  PROC DrawPart84()
    MoveL Offs(pOrigin,162.64,96.16,0.00),v40,z0,tPen\WObj:=wPaper;
    MoveL Offs(pOrigin,162.24,96.31,0.00),v40,z0,tPen\WObj:=wPaper;
    MoveL Offs(pOrigin,173.08,96.31,0.00),v40,z0,tPen\WObj:=wPaper;
    MoveL Offs(pOrigin,173.29,96.59,0.00),v40,z0,tPen\WObj:=wPaper;
    MoveL Offs(pOrigin,180.51,104.24,0.00),v40,z0,tPen\WObj:=wPaper;
    MoveL Offs(pOrigin,193.05,116.56,0.00),v40,fine,tPen\WObj:=wPaper;
    MoveL Offs(pOrigin,193.05,116.56,6.00),v60,z5,tPen\WObj:=wPaper;
    MoveL Offs(pOrigin,193.92,115.46,6.00),vTravel,z5,tPen\WObj:=wPaper;
    MoveL Offs(pOrigin,193.92,115.46,0.00),v60,z0,tPen\WObj:=wPaper;
    MoveL Offs(pOrigin,194.97,114.41,0.00),v40,z0,tPen\WObj:=wPaper;
    MoveL Offs(pOrigin,195.87,115.01,0.00),v40,z0,tPen\WObj:=wPaper;
    MoveL Offs(pOrigin,194.82,116.06,0.00),v40,z0,tPen\WObj:=wPaper;
    MoveL Offs(pOrigin,195.71,116.66,0.00),v40,z0,tPen\WObj:=wPaper;
    MoveL Offs(pOrigin,196.47,115.91,0.00),v40,fine,tPen\WObj:=wPaper;
    MoveL Offs(pOrigin,196.47,115.91,6.00),v60,z5,tPen\WObj:=wPaper;
    MoveL Offs(pOrigin,194.38,113.52,6.00),vTravel,z5,tPen\WObj:=wPaper;
    MoveL Offs(pOrigin,194.38,113.52,0.00),v60,z0,tPen\WObj:=wPaper;
    MoveL Offs(pOrigin,193.02,114.87,0.00),v40,z0,tPen\WObj:=wPaper;
    MoveL Offs(pOrigin,193.69,114.22,0.00),v40,z0,tPen\WObj:=wPaper;
    MoveL Offs(pOrigin,194.11,114.65,0.00),v40,z0,tPen\WObj:=wPaper;
    MoveL Offs(pOrigin,193.69,114.22,0.00),v40,fine,tPen\WObj:=wPaper;
    MoveL Offs(pOrigin,193.69,114.22,6.00),v60,z5,tPen\WObj:=wPaper;
    MoveL Offs(pOrigin,193.48,112.92,6.00),vTravel,z5,tPen\WObj:=wPaper;
    MoveL Offs(pOrigin,193.48,112.92,0.00),v60,z0,tPen\WObj:=wPaper;
    MoveL Offs(pOrigin,191.68,114.72,0.00),v40,z0,tPen\WObj:=wPaper;
    MoveL Offs(pOrigin,190.63,114.28,0.00),v40,z0,tPen\WObj:=wPaper;
    MoveL Offs(pOrigin,192.88,112.02,0.00),v40,z0,tPen\WObj:=wPaper;
    MoveL Offs(pOrigin,191.99,111.43,0.00),v40,z0,tPen\WObj:=wPaper;
    MoveL Offs(pOrigin,189.88,113.53,0.00),v40,z0,tPen\WObj:=wPaper;
    MoveL Offs(pOrigin,188.98,112.93,0.00),v40,z0,tPen\WObj:=wPaper;
    MoveL Offs(pOrigin,191.39,110.53,0.00),v40,z0,tPen\WObj:=wPaper;
    MoveL Offs(pOrigin,190.64,109.78,0.00),v40,z0,tPen\WObj:=wPaper;
    MoveL Offs(pOrigin,188.09,112.34,0.00),v40,z0,tPen\WObj:=wPaper;
    MoveL Offs(pOrigin,187.34,111.59,0.00),v40,z0,tPen\WObj:=wPaper;
    MoveL Offs(pOrigin,189.90,109.04,0.00),v40,z0,tPen\WObj:=wPaper;
    MoveL Offs(pOrigin,189.15,108.29,0.00),v40,z0,tPen\WObj:=wPaper;
    MoveL Offs(pOrigin,186.44,110.99,0.00),v40,z0,tPen\WObj:=wPaper;
    MoveL Offs(pOrigin,186.46,109.97,0.00),v40,z0,tPen\WObj:=wPaper;
    MoveL Offs(pOrigin,186.89,110.40,0.00),v40,z0,tPen\WObj:=wPaper;
    MoveL Offs(pOrigin,186.46,109.97,0.00),v40,z0,tPen\WObj:=wPaper;
    MoveL Offs(pOrigin,185.70,110.25,0.00),v40,z0,tPen\WObj:=wPaper;
    MoveL Offs(pOrigin,188.55,107.39,0.00),v40,z0,tPen\WObj:=wPaper;
    MoveL Offs(pOrigin,187.81,106.65,0.00),v40,z0,tPen\WObj:=wPaper;
    MoveL Offs(pOrigin,184.95,109.50,0.00),v40,z0,tPen\WObj:=wPaper;
    MoveL Offs(pOrigin,184.20,108.75,0.00),v40,z0,tPen\WObj:=wPaper;
    MoveL Offs(pOrigin,187.21,105.75,0.00),v40,z0,tPen\WObj:=wPaper;
    MoveL Offs(pOrigin,186.46,105.00,0.00),v40,z0,tPen\WObj:=wPaper;
    MoveL Offs(pOrigin,183.31,108.16,0.00),v40,z0,tPen\WObj:=wPaper;
    MoveL Offs(pOrigin,183.70,107.21,0.00),v40,z0,tPen\WObj:=wPaper;
    MoveL Offs(pOrigin,184.55,108.06,0.00),v40,z0,tPen\WObj:=wPaper;
    MoveL Offs(pOrigin,183.70,107.21,0.00),v40,z0,tPen\WObj:=wPaper;
    MoveL Offs(pOrigin,182.71,107.26,0.00),v40,z0,tPen\WObj:=wPaper;
    MoveL Offs(pOrigin,185.87,104.10,0.00),v40,z0,tPen\WObj:=wPaper;
    MoveL Offs(pOrigin,185.27,103.21,0.00),v40,z0,tPen\WObj:=wPaper;
    MoveL Offs(pOrigin,181.81,106.66,0.00),v40,z0,tPen\WObj:=wPaper;
    MoveL Offs(pOrigin,182.21,105.72,0.00),v40,z0,tPen\WObj:=wPaper;
    MoveL Offs(pOrigin,183.06,106.57,0.00),v40,z0,tPen\WObj:=wPaper;
    MoveL Offs(pOrigin,182.21,105.72,0.00),v40,z0,tPen\WObj:=wPaper;
    MoveL Offs(pOrigin,181.07,105.92,0.00),v40,z0,tPen\WObj:=wPaper;
    MoveL Offs(pOrigin,182.42,104.56,0.00),v40,z0,tPen\WObj:=wPaper;
    MoveL Offs(pOrigin,181.67,103.82,0.00),v40,z0,tPen\WObj:=wPaper;
    MoveL Offs(pOrigin,180.32,105.17,0.00),v40,z0,tPen\WObj:=wPaper;
    MoveL Offs(pOrigin,181.15,104.66,0.00),v40,z0,tPen\WObj:=wPaper;
    MoveL Offs(pOrigin,182.00,105.51,0.00),v40,z0,tPen\WObj:=wPaper;
    MoveL Offs(pOrigin,181.15,104.66,0.00),v40,fine,tPen\WObj:=wPaper;
    MoveL Offs(pOrigin,181.15,104.66,6.00),v60,z5,tPen\WObj:=wPaper;
    MoveL Offs(pOrigin,179.57,104.42,6.00),vTravel,z5,tPen\WObj:=wPaper;
    MoveL Offs(pOrigin,179.57,104.42,0.00),v60,z0,tPen\WObj:=wPaper;
    MoveL Offs(pOrigin,180.93,103.07,0.00),v40,z0,tPen\WObj:=wPaper;
    MoveL Offs(pOrigin,180.18,102.32,0.00),v40,z0,tPen\WObj:=wPaper;
    MoveL Offs(pOrigin,178.83,103.68,0.00),v40,z0,tPen\WObj:=wPaper;
    MoveL Offs(pOrigin,179.59,103.72,0.00),v40,z0,tPen\WObj:=wPaper;
    MoveL Offs(pOrigin,175.68,99.81,0.00),v40,z0,tPen\WObj:=wPaper;
    MoveL Offs(pOrigin,175.09,99.94,0.00),v40,z0,tPen\WObj:=wPaper;
    MoveL Offs(pOrigin,176.60,98.44,0.00),v40,z0,tPen\WObj:=wPaper;
    MoveL Offs(pOrigin,175.84,99.14,0.00),v40,z0,tPen\WObj:=wPaper;
    MoveL Offs(pOrigin,176.26,99.56,0.00),v40,z0,tPen\WObj:=wPaper;
    MoveL Offs(pOrigin,175.84,99.14,0.00),v40,fine,tPen\WObj:=wPaper;
    MoveL Offs(pOrigin,175.84,99.14,6.00),v60,z5,tPen\WObj:=wPaper;
    MoveL Offs(pOrigin,174.50,99.05,6.00),vTravel,z5,tPen\WObj:=wPaper;
    MoveL Offs(pOrigin,174.50,99.05,0.00),v60,z0,tPen\WObj:=wPaper;
    MoveL Offs(pOrigin,175.85,97.69,0.00),v40,z0,tPen\WObj:=wPaper;
    MoveL Offs(pOrigin,175.10,96.95,0.00),v40,z0,tPen\WObj:=wPaper;
    MoveL Offs(pOrigin,173.60,98.45,0.00),v40,z0,tPen\WObj:=wPaper;
    MoveL Offs(pOrigin,173.00,97.55,0.00),v40,z0,tPen\WObj:=wPaper;
    MoveL Offs(pOrigin,202.60,67.95,0.00),v40,z0,tPen\WObj:=wPaper;
    MoveL Offs(pOrigin,203.75,68.14,0.00),v40,z0,tPen\WObj:=wPaper;
    MoveL Offs(pOrigin,205.55,69.94,0.00),v40,z0,tPen\WObj:=wPaper;
    MoveL Offs(pOrigin,205.80,69.60,0.00),v40,z0,tPen\WObj:=wPaper;
    MoveL Offs(pOrigin,206.23,68.75,0.00),v40,z0,tPen\WObj:=wPaper;
    MoveL Offs(pOrigin,214.51,62.52,0.00),v40,z0,tPen\WObj:=wPaper;
    MoveL Offs(pOrigin,214.73,63.22,0.00),v40,z0,tPen\WObj:=wPaper;
    MoveL Offs(pOrigin,214.30,68.96,0.00),v40,z0,tPen\WObj:=wPaper;
    MoveL Offs(pOrigin,213.95,70.24,0.00),v40,z0,tPen\WObj:=wPaper;
    MoveL Offs(pOrigin,213.02,71.51,0.00),v40,z0,tPen\WObj:=wPaper;
    MoveL Offs(pOrigin,212.59,71.01,0.00),v40,z0,tPen\WObj:=wPaper;
    MoveL Offs(pOrigin,214.40,72.82,0.00),v40,z0,tPen\WObj:=wPaper;
    MoveL Offs(pOrigin,214.09,72.57,0.00),v40,z0,tPen\WObj:=wPaper;
    MoveL Offs(pOrigin,215.01,71.30,0.00),v40,z0,tPen\WObj:=wPaper;
    MoveL Offs(pOrigin,215.86,68.61,0.00),v40,z0,tPen\WObj:=wPaper;
    MoveL Offs(pOrigin,216.21,68.54,0.00),v40,z0,tPen\WObj:=wPaper;
    MoveL Offs(pOrigin,216.21,68.54,0.00),v40,z0,tPen\WObj:=wPaper;
    MoveL Offs(pOrigin,216.00,64.93,0.00),v40,z0,tPen\WObj:=wPaper;
    MoveL Offs(pOrigin,216.21,63.86,0.00),v40,fine,tPen\WObj:=wPaper;
    MoveL Offs(pOrigin,216.21,63.86,6.00),v60,z5,tPen\WObj:=wPaper;
    MoveL Offs(pOrigin,217.49,63.58,6.00),vTravel,z5,tPen\WObj:=wPaper;
    MoveL Offs(pOrigin,217.49,63.58,0.00),v60,z0,tPen\WObj:=wPaper;
    MoveL Offs(pOrigin,214.51,63.58,0.00),v40,z0,tPen\WObj:=wPaper;
    MoveL Offs(pOrigin,214.38,62.59,0.00),v40,z0,tPen\WObj:=wPaper;
    MoveL Offs(pOrigin,214.38,60.89,0.00),v40,z0,tPen\WObj:=wPaper;
    MoveL Offs(pOrigin,214.30,60.46,0.00),v40,z0,tPen\WObj:=wPaper;
    MoveL Offs(pOrigin,213.24,61.53,0.00),v40,z0,tPen\WObj:=wPaper;
    MoveL Offs(pOrigin,214.30,60.46,0.00),v40,z0,tPen\WObj:=wPaper;
    MoveL Offs(pOrigin,214.51,60.41,0.00),v40,z0,tPen\WObj:=wPaper;
    MoveL Offs(pOrigin,217.28,60.41,0.00),v40,z0,tPen\WObj:=wPaper;
    MoveL Offs(pOrigin,218.06,59.96,0.00),v40,z0,tPen\WObj:=wPaper;
    MoveL Offs(pOrigin,212.95,65.07,0.00),v40,z0,tPen\WObj:=wPaper;
    MoveL Offs(pOrigin,212.12,64.57,0.00),v40,z0,tPen\WObj:=wPaper;
    MoveL Offs(pOrigin,210.77,63.22,0.00),v40,z0,tPen\WObj:=wPaper;
    MoveL Offs(pOrigin,211.11,63.58,0.00),v40,z0,tPen\WObj:=wPaper;
  ENDPROC

  PROC DrawPart85()
    MoveL Offs(pOrigin,212.60,63.58,0.00),v40,z0,tPen\WObj:=wPaper;
    MoveL Offs(pOrigin,212.39,62.52,0.00),v40,z0,tPen\WObj:=wPaper;
    MoveL Offs(pOrigin,217.49,62.52,0.00),v40,z0,tPen\WObj:=wPaper;
    MoveL Offs(pOrigin,217.96,62.94,0.00),v40,z0,tPen\WObj:=wPaper;
    MoveL Offs(pOrigin,214.51,59.48,0.00),v40,z0,tPen\WObj:=wPaper;
    MoveL Offs(pOrigin,214.94,59.19,0.00),v40,z0,tPen\WObj:=wPaper;
    MoveL Offs(pOrigin,213.66,58.76,0.00),v40,z0,tPen\WObj:=wPaper;
    MoveL Offs(pOrigin,212.46,56.64,0.00),v40,z0,tPen\WObj:=wPaper;
    MoveL Offs(pOrigin,212.18,54.72,0.00),v40,z0,tPen\WObj:=wPaper;
    MoveL Offs(pOrigin,212.60,53.88,0.00),v40,z0,tPen\WObj:=wPaper;
    MoveL Offs(pOrigin,212.99,53.49,0.00),v40,z0,tPen\WObj:=wPaper;
    MoveL Offs(pOrigin,211.04,51.53,0.00),v40,z0,tPen\WObj:=wPaper;
    MoveL Offs(pOrigin,211.32,51.96,0.00),v40,z0,tPen\WObj:=wPaper;
    MoveL Offs(pOrigin,215.58,51.96,0.00),v40,fine,tPen\WObj:=wPaper;
    MoveL Offs(pOrigin,215.58,51.96,6.00),v60,z5,tPen\WObj:=wPaper;
    MoveL Offs(pOrigin,216.49,52.81,6.00),vTravel,z5,tPen\WObj:=wPaper;
    MoveL Offs(pOrigin,216.49,52.81,0.00),v60,z0,tPen\WObj:=wPaper;
    MoveL Offs(pOrigin,216.49,54.30,0.00),v40,z0,tPen\WObj:=wPaper;
    MoveL Offs(pOrigin,215.79,54.07,0.00),v40,z0,tPen\WObj:=wPaper;
    MoveL Offs(pOrigin,218.12,54.07,0.00),v40,z0,tPen\WObj:=wPaper;
    MoveL Offs(pOrigin,217.55,53.88,0.00),v40,z0,tPen\WObj:=wPaper;
    MoveL Offs(pOrigin,217.55,52.60,0.00),v40,z0,tPen\WObj:=wPaper;
    MoveL Offs(pOrigin,217.28,51.96,0.00),v40,z0,tPen\WObj:=wPaper;
    MoveL Offs(pOrigin,219.82,51.96,0.00),v40,z0,tPen\WObj:=wPaper;
    MoveL Offs(pOrigin,219.61,52.17,0.00),v40,z0,tPen\WObj:=wPaper;
    MoveL Offs(pOrigin,219.19,52.60,0.00),v40,z0,tPen\WObj:=wPaper;
    MoveL Offs(pOrigin,219.61,52.17,0.00),v40,z0,tPen\WObj:=wPaper;
    MoveL Offs(pOrigin,219.73,52.76,0.00),v40,z0,tPen\WObj:=wPaper;
    MoveL Offs(pOrigin,217.77,50.81,0.00),v40,z0,tPen\WObj:=wPaper;
    MoveL Offs(pOrigin,218.34,50.90,0.00),v40,z0,tPen\WObj:=wPaper;
    MoveL Offs(pOrigin,222.80,50.90,0.00),v40,z0,tPen\WObj:=wPaper;
    MoveL Offs(pOrigin,223.01,50.07,0.00),v40,z0,tPen\WObj:=wPaper;
    MoveL Offs(pOrigin,220.61,47.67,0.00),v40,z0,tPen\WObj:=wPaper;
    MoveL Offs(pOrigin,221.31,47.74,0.00),v40,z0,tPen\WObj:=wPaper;
    MoveL Offs(pOrigin,223.22,47.74,0.00),v40,z0,tPen\WObj:=wPaper;
    MoveL Offs(pOrigin,223.44,47.71,0.00),v40,z0,tPen\WObj:=wPaper;
    MoveL Offs(pOrigin,223.01,48.35,0.00),v40,z0,tPen\WObj:=wPaper;
    MoveL Offs(pOrigin,223.44,47.71,0.00),v40,z0,tPen\WObj:=wPaper;
    MoveL Offs(pOrigin,223.76,47.83,0.00),v40,z0,tPen\WObj:=wPaper;
    MoveL Offs(pOrigin,216.54,40.62,0.00),v40,z0,tPen\WObj:=wPaper;
    MoveL Offs(pOrigin,215.57,40.05,0.00),v40,z0,tPen\WObj:=wPaper;
    MoveL Offs(pOrigin,211.52,44.11,0.00),v40,z0,tPen\WObj:=wPaper;
    MoveL Offs(pOrigin,210.56,43.59,0.00),v40,z0,tPen\WObj:=wPaper;
    MoveL Offs(pOrigin,199.59,32.62,0.00),v40,z0,tPen\WObj:=wPaper;
    MoveL Offs(pOrigin,200.06,32.95,0.00),v40,z0,tPen\WObj:=wPaper;
    MoveL Offs(pOrigin,195.39,32.95,0.00),v40,fine,tPen\WObj:=wPaper;
    MoveL Offs(pOrigin,195.39,32.95,6.00),v60,z5,tPen\WObj:=wPaper;
    MoveL Offs(pOrigin,196.02,31.90,6.00),vTravel,z5,tPen\WObj:=wPaper;
    MoveL Offs(pOrigin,196.02,31.90,0.00),v60,z0,tPen\WObj:=wPaper;
    MoveL Offs(pOrigin,166.70,31.90,0.00),v40,z0,tPen\WObj:=wPaper;
    MoveL Offs(pOrigin,167.23,31.63,0.00),v40,z0,tPen\WObj:=wPaper;
    MoveL Offs(pOrigin,168.89,33.28,0.00),v40,z0,tPen\WObj:=wPaper;
    MoveL Offs(pOrigin,168.11,33.75,0.00),v40,z0,tPen\WObj:=wPaper;
    MoveL Offs(pOrigin,171.11,30.75,0.00),v40,z0,tPen\WObj:=wPaper;
    MoveL Offs(pOrigin,171.28,31.19,0.00),v40,z0,tPen\WObj:=wPaper;
    MoveL Offs(pOrigin,173.08,32.99,0.00),v40,z0,tPen\WObj:=wPaper;
    MoveL Offs(pOrigin,172.90,33.44,0.00),v40,z0,tPen\WObj:=wPaper;
    MoveL Offs(pOrigin,175.61,30.73,0.00),v40,z0,tPen\WObj:=wPaper;
    MoveL Offs(pOrigin,175.62,31.05,0.00),v40,z0,tPen\WObj:=wPaper;
    MoveL Offs(pOrigin,177.87,33.31,0.00),v40,z0,tPen\WObj:=wPaper;
    MoveL Offs(pOrigin,176.94,33.88,0.00),v40,z0,tPen\WObj:=wPaper;
    MoveL Offs(pOrigin,180.10,30.72,0.00),v40,z0,tPen\WObj:=wPaper;
    MoveL Offs(pOrigin,180.41,31.37,0.00),v40,z0,tPen\WObj:=wPaper;
    MoveL Offs(pOrigin,181.92,32.87,0.00),v40,z0,tPen\WObj:=wPaper;
    MoveL Offs(pOrigin,182.04,33.26,0.00),v40,z0,tPen\WObj:=wPaper;
    MoveL Offs(pOrigin,184.89,30.41,0.00),v40,z0,tPen\WObj:=wPaper;
    MoveL Offs(pOrigin,184.46,30.93,0.00),v40,z0,tPen\WObj:=wPaper;
    MoveL Offs(pOrigin,186.26,32.73,0.00),v40,z0,tPen\WObj:=wPaper;
    MoveL Offs(pOrigin,186.53,33.25,0.00),v40,z0,tPen\WObj:=wPaper;
    MoveL Offs(pOrigin,189.39,30.39,0.00),v40,z0,tPen\WObj:=wPaper;
    MoveL Offs(pOrigin,188.95,30.94,0.00),v40,z0,tPen\WObj:=wPaper;
    MoveL Offs(pOrigin,190.90,32.90,0.00),v40,z0,tPen\WObj:=wPaper;
    MoveL Offs(pOrigin,191.03,33.23,0.00),v40,z0,tPen\WObj:=wPaper;
    MoveL Offs(pOrigin,193.58,30.68,0.00),v40,z0,tPen\WObj:=wPaper;
    MoveL Offs(pOrigin,193.90,31.41,0.00),v40,z0,tPen\WObj:=wPaper;
    MoveL Offs(pOrigin,199.91,37.42,0.00),v40,z0,tPen\WObj:=wPaper;
    MoveL Offs(pOrigin,199.85,37.85,0.00),v40,z0,tPen\WObj:=wPaper;
    MoveL Offs(pOrigin,205.86,31.84,0.00),v40,fine,tPen\WObj:=wPaper;
    MoveL Offs(pOrigin,205.86,31.84,6.00),v60,z5,tPen\WObj:=wPaper;
    MoveL Offs(pOrigin,204.36,31.84,6.00),vTravel,z5,tPen\WObj:=wPaper;
    MoveL Offs(pOrigin,204.36,31.84,0.00),v60,z0,tPen\WObj:=wPaper;
    MoveL Offs(pOrigin,198.50,37.70,0.00),v40,z0,tPen\WObj:=wPaper;
    MoveL Offs(pOrigin,198.11,37.11,0.00),v40,z0,tPen\WObj:=wPaper;
    MoveL Offs(pOrigin,196.46,35.46,0.00),v40,fine,tPen\WObj:=wPaper;
    MoveL Offs(pOrigin,196.46,35.46,6.00),v60,z5,tPen\WObj:=wPaper;
    MoveL Offs(pOrigin,194.96,35.46,6.00),vTravel,z5,tPen\WObj:=wPaper;
    MoveL Offs(pOrigin,194.96,35.46,0.00),v60,z0,tPen\WObj:=wPaper;
    MoveL Offs(pOrigin,196.61,37.11,0.00),v40,z0,tPen\WObj:=wPaper;
    MoveL Offs(pOrigin,197.01,37.71,0.00),v40,z0,tPen\WObj:=wPaper;
    MoveL Offs(pOrigin,202.87,31.85,0.00),v40,fine,tPen\WObj:=wPaper;
    MoveL Offs(pOrigin,202.87,31.85,6.00),v60,z5,tPen\WObj:=wPaper;
    MoveL Offs(pOrigin,200.49,33.26,6.00),vTravel,z5,tPen\WObj:=wPaper;
    MoveL Offs(pOrigin,200.49,33.26,0.00),v60,z0,tPen\WObj:=wPaper;
    MoveL Offs(pOrigin,201.55,34.75,0.00),v40,z0,tPen\WObj:=wPaper;
    MoveL Offs(pOrigin,203.04,35.39,0.00),v40,z0,tPen\WObj:=wPaper;
    MoveL Offs(pOrigin,210.48,34.75,0.00),v40,z0,tPen\WObj:=wPaper;
    MoveL Offs(pOrigin,235.12,33.69,0.00),v40,z0,tPen\WObj:=wPaper;
    MoveL Offs(pOrigin,237.68,33.26,0.00),v40,fine,tPen\WObj:=wPaper;
    MoveL Offs(pOrigin,237.68,33.26,6.00),v60,z5,tPen\WObj:=wPaper;
    MoveL Offs(pOrigin,240.75,35.78,6.00),vTravel,z5,tPen\WObj:=wPaper;
    MoveL Offs(pOrigin,240.75,35.78,0.00),v60,z0,tPen\WObj:=wPaper;
    MoveL Offs(pOrigin,248.87,27.66,0.00),v40,z0,tPen\WObj:=wPaper;
    MoveL Offs(pOrigin,249.16,28.43,0.00),v40,z0,tPen\WObj:=wPaper;
    MoveL Offs(pOrigin,254.72,33.99,0.00),v40,z0,tPen\WObj:=wPaper;
    MoveL Offs(pOrigin,255.29,34.68,0.00),v40,z0,tPen\WObj:=wPaper;
    MoveL Offs(pOrigin,257.39,32.58,0.00),v40,fine,tPen\WObj:=wPaper;
    MoveL Offs(pOrigin,257.39,32.58,6.00),v60,z5,tPen\WObj:=wPaper;
    MoveL Offs(pOrigin,255.31,32.20,6.00),vTravel,z5,tPen\WObj:=wPaper;
    MoveL Offs(pOrigin,255.31,32.20,0.00),v60,z0,tPen\WObj:=wPaper;
    MoveL Offs(pOrigin,256.16,33.05,0.00),v40,z0,tPen\WObj:=wPaper;
    MoveL Offs(pOrigin,255.31,32.20,0.00),v40,fine,tPen\WObj:=wPaper;
    MoveL Offs(pOrigin,255.31,32.20,6.00),v60,z5,tPen\WObj:=wPaper;
    MoveL Offs(pOrigin,253.45,31.99,6.00),vTravel,z5,tPen\WObj:=wPaper;
    MoveL Offs(pOrigin,253.45,31.99,0.00),v60,z0,tPen\WObj:=wPaper;
    MoveL Offs(pOrigin,253.45,30.29,0.00),v40,fine,tPen\WObj:=wPaper;
    MoveL Offs(pOrigin,253.45,30.29,6.00),v60,z5,tPen\WObj:=wPaper;
    MoveL Offs(pOrigin,255.95,30.08,6.00),vTravel,z5,tPen\WObj:=wPaper;
    MoveL Offs(pOrigin,255.95,30.08,0.00),v60,z0,tPen\WObj:=wPaper;
    MoveL Offs(pOrigin,255.52,30.50,0.00),v40,z0,tPen\WObj:=wPaper;
    MoveL Offs(pOrigin,255.95,30.08,0.00),v40,z0,tPen\WObj:=wPaper;
  ENDPROC

  PROC DrawPart86()
    MoveL Offs(pOrigin,256.16,29.78,0.00),v40,z0,tPen\WObj:=wPaper;
    MoveL Offs(pOrigin,247.02,29.78,0.00),v40,fine,tPen\WObj:=wPaper;
    MoveL Offs(pOrigin,247.02,29.78,6.00),v60,z5,tPen\WObj:=wPaper;
    MoveL Offs(pOrigin,247.88,28.73,6.00),vTravel,z5,tPen\WObj:=wPaper;
    MoveL Offs(pOrigin,247.88,28.73,0.00),v60,z0,tPen\WObj:=wPaper;
    MoveL Offs(pOrigin,249.79,28.73,0.00),v40,z0,tPen\WObj:=wPaper;
    MoveL Offs(pOrigin,250.29,29.44,0.00),v40,z0,tPen\WObj:=wPaper;
    MoveL Offs(pOrigin,250.29,30.92,0.00),v40,z0,tPen\WObj:=wPaper;
    MoveL Offs(pOrigin,249.23,30.71,0.00),v40,z0,tPen\WObj:=wPaper;
    MoveL Offs(pOrigin,249.23,29.44,0.00),v40,fine,tPen\WObj:=wPaper;
    MoveL Offs(pOrigin,249.23,29.44,6.00),v60,z5,tPen\WObj:=wPaper;
    MoveL Offs(pOrigin,250.21,27.81,6.00),vTravel,z5,tPen\WObj:=wPaper;
    MoveL Offs(pOrigin,250.21,27.81,0.00),v60,z0,tPen\WObj:=wPaper;
    MoveL Offs(pOrigin,236.54,41.48,0.00),v40,z0,tPen\WObj:=wPaper;
    MoveL Offs(pOrigin,236.47,41.13,0.00),v40,z0,tPen\WObj:=wPaper;
    MoveL Offs(pOrigin,234.52,39.17,0.00),v40,z0,tPen\WObj:=wPaper;
    MoveL Offs(pOrigin,235.05,38.49,0.00),v40,z0,tPen\WObj:=wPaper;
    MoveL Offs(pOrigin,231.90,41.65,0.00),v40,z0,tPen\WObj:=wPaper;
    MoveL Offs(pOrigin,232.43,41.56,0.00),v40,z0,tPen\WObj:=wPaper;
    MoveL Offs(pOrigin,230.47,39.61,0.00),v40,fine,tPen\WObj:=wPaper;
    MoveL Offs(pOrigin,230.47,39.61,6.00),v60,z5,tPen\WObj:=wPaper;
    MoveL Offs(pOrigin,228.97,39.60,6.00),vTravel,z5,tPen\WObj:=wPaper;
    MoveL Offs(pOrigin,228.97,39.60,0.00),v60,z0,tPen\WObj:=wPaper;
    MoveL Offs(pOrigin,230.93,41.56,0.00),v40,z0,tPen\WObj:=wPaper;
    MoveL Offs(pOrigin,230.10,41.95,0.00),v40,z0,tPen\WObj:=wPaper;
    MoveL Offs(pOrigin,233.55,38.50,0.00),v40,z0,tPen\WObj:=wPaper;
    MoveL Offs(pOrigin,233.02,39.17,0.00),v40,z0,tPen\WObj:=wPaper;
    MoveL Offs(pOrigin,234.97,41.12,0.00),v40,z0,tPen\WObj:=wPaper;
    MoveL Offs(pOrigin,235.04,41.49,0.00),v40,z0,tPen\WObj:=wPaper;
    MoveL Offs(pOrigin,238.35,38.18,0.00),v40,fine,tPen\WObj:=wPaper;
    MoveL Offs(pOrigin,238.35,38.18,6.00),v60,z5,tPen\WObj:=wPaper;
    MoveL Offs(pOrigin,241.25,36.95,6.00),vTravel,z5,tPen\WObj:=wPaper;
    MoveL Offs(pOrigin,241.25,36.95,0.00),v60,z0,tPen\WObj:=wPaper;
    MoveL Offs(pOrigin,244.10,39.80,0.00),v40,z0,tPen\WObj:=wPaper;
    MoveL Offs(pOrigin,244.49,39.51,0.00),v40,z0,tPen\WObj:=wPaper;
    MoveL Offs(pOrigin,242.08,41.92,0.00),v40,z0,tPen\WObj:=wPaper;
    MoveL Offs(pOrigin,242.68,42.81,0.00),v40,z0,tPen\WObj:=wPaper;
    MoveL Offs(pOrigin,245.08,40.41,0.00),v40,z0,tPen\WObj:=wPaper;
    MoveL Offs(pOrigin,244.05,40.34,0.00),v40,z0,tPen\WObj:=wPaper;
    MoveL Offs(pOrigin,241.71,40.34,0.00),v40,z0,tPen\WObj:=wPaper;
    MoveL Offs(pOrigin,241.84,40.06,0.00),v40,z0,tPen\WObj:=wPaper;
    MoveL Offs(pOrigin,241.84,38.15,0.00),v40,z0,tPen\WObj:=wPaper;
    MoveL Offs(pOrigin,241.50,37.18,0.00),v40,z0,tPen\WObj:=wPaper;
    MoveL Offs(pOrigin,242.78,37.18,0.00),v40,fine,tPen\WObj:=wPaper;
    MoveL Offs(pOrigin,242.78,37.18,6.00),v60,z5,tPen\WObj:=wPaper;
    MoveL Offs(pOrigin,246.39,36.24,6.00),vTravel,z5,tPen\WObj:=wPaper;
    MoveL Offs(pOrigin,246.39,36.24,0.00),v60,z0,tPen\WObj:=wPaper;
    MoveL Offs(pOrigin,246.81,36.66,0.00),v40,z0,tPen\WObj:=wPaper;
    MoveL Offs(pOrigin,246.39,36.24,0.00),v40,z0,tPen\WObj:=wPaper;
    MoveL Offs(pOrigin,246.89,35.61,0.00),v40,z0,tPen\WObj:=wPaper;
    MoveL Offs(pOrigin,241.18,41.32,0.00),v40,fine,tPen\WObj:=wPaper;
    MoveL Offs(pOrigin,241.18,41.32,6.00),v60,z5,tPen\WObj:=wPaper;
    MoveL Offs(pOrigin,243.84,42.46,6.00),vTravel,z5,tPen\WObj:=wPaper;
    MoveL Offs(pOrigin,243.84,42.46,0.00),v60,z0,tPen\WObj:=wPaper;
    MoveL Offs(pOrigin,245.54,42.46,0.00),v40,fine,tPen\WObj:=wPaper;
    MoveL Offs(pOrigin,245.54,42.46,6.00),v60,z5,tPen\WObj:=wPaper;
    MoveL Offs(pOrigin,246.81,44.53,6.00),vTravel,z5,tPen\WObj:=wPaper;
    MoveL Offs(pOrigin,246.81,44.53,0.00),v60,z0,tPen\WObj:=wPaper;
    MoveL Offs(pOrigin,248.09,45.80,0.00),v40,z0,tPen\WObj:=wPaper;
    MoveL Offs(pOrigin,246.81,44.53,0.00),v40,z0,tPen\WObj:=wPaper;
    MoveL Offs(pOrigin,246.39,45.62,0.00),v40,z0,tPen\WObj:=wPaper;
    MoveL Offs(pOrigin,247.88,45.62,0.00),v40,z0,tPen\WObj:=wPaper;
    MoveL Offs(pOrigin,247.45,46.68,0.00),v40,z0,tPen\WObj:=wPaper;
    MoveL Offs(pOrigin,248.94,46.68,0.00),v40,z0,tPen\WObj:=wPaper;
    MoveL Offs(pOrigin,249.36,47.29,0.00),v40,z0,tPen\WObj:=wPaper;
    MoveL Offs(pOrigin,250.21,48.14,0.00),v40,z0,tPen\WObj:=wPaper;
    MoveL Offs(pOrigin,249.36,47.29,0.00),v40,z0,tPen\WObj:=wPaper;
    MoveL Offs(pOrigin,250.00,47.74,0.00),v40,z0,tPen\WObj:=wPaper;
    MoveL Offs(pOrigin,248.30,47.74,0.00),v40,z0,tPen\WObj:=wPaper;
    MoveL Offs(pOrigin,247.45,47.29,0.00),v40,z0,tPen\WObj:=wPaper;
    MoveL Offs(pOrigin,248.30,48.14,0.00),v40,z0,tPen\WObj:=wPaper;
    MoveL Offs(pOrigin,247.45,47.29,0.00),v40,fine,tPen\WObj:=wPaper;
    MoveL Offs(pOrigin,247.45,47.29,6.00),v60,z5,tPen\WObj:=wPaper;
    MoveL Offs(pOrigin,246.18,45.80,6.00),vTravel,z5,tPen\WObj:=wPaper;
    MoveL Offs(pOrigin,246.18,45.80,0.00),v60,z0,tPen\WObj:=wPaper;
    MoveL Offs(pOrigin,246.60,46.22,0.00),v40,z0,tPen\WObj:=wPaper;
    MoveL Offs(pOrigin,246.18,45.80,0.00),v40,fine,tPen\WObj:=wPaper;
    MoveL Offs(pOrigin,246.18,45.80,6.00),v60,z5,tPen\WObj:=wPaper;
    MoveL Offs(pOrigin,249.36,48.79,6.00),vTravel,z5,tPen\WObj:=wPaper;
    MoveL Offs(pOrigin,249.36,48.79,0.00),v60,z0,tPen\WObj:=wPaper;
    MoveL Offs(pOrigin,250.85,48.79,0.00),v40,z0,tPen\WObj:=wPaper;
    MoveL Offs(pOrigin,250.43,48.35,0.00),v40,z0,tPen\WObj:=wPaper;
    MoveL Offs(pOrigin,250.64,48.78,0.00),v40,z0,tPen\WObj:=wPaper;
    MoveL Offs(pOrigin,250.43,48.35,0.00),v40,fine,tPen\WObj:=wPaper;
    MoveL Offs(pOrigin,250.43,48.35,6.00),v60,z5,tPen\WObj:=wPaper;
    MoveL Offs(pOrigin,251.70,49.84,6.00),vTravel,z5,tPen\WObj:=wPaper;
    MoveL Offs(pOrigin,251.70,49.84,0.00),v60,z0,tPen\WObj:=wPaper;
    MoveL Offs(pOrigin,253.19,51.33,0.00),v40,z0,tPen\WObj:=wPaper;
    MoveL Offs(pOrigin,251.70,49.84,0.00),v40,fine,tPen\WObj:=wPaper;
    MoveL Offs(pOrigin,251.70,49.84,6.00),v60,z5,tPen\WObj:=wPaper;
    MoveL Offs(pOrigin,253.44,49.97,6.00),vTravel,z5,tPen\WObj:=wPaper;
    MoveL Offs(pOrigin,253.44,49.97,0.00),v60,z0,tPen\WObj:=wPaper;
    MoveL Offs(pOrigin,251.04,52.37,0.00),v40,fine,tPen\WObj:=wPaper;
    MoveL Offs(pOrigin,251.04,52.37,6.00),v60,z5,tPen\WObj:=wPaper;
    MoveL Offs(pOrigin,254.02,55.36,6.00),vTravel,z5,tPen\WObj:=wPaper;
    MoveL Offs(pOrigin,254.02,55.36,0.00),v60,z0,tPen\WObj:=wPaper;
    MoveL Offs(pOrigin,256.43,52.96,0.00),v40,fine,tPen\WObj:=wPaper;
    MoveL Offs(pOrigin,256.43,52.96,6.00),v60,z5,tPen\WObj:=wPaper;
    MoveL Offs(pOrigin,262.28,51.59,6.00),vTravel,z5,tPen\WObj:=wPaper;
    MoveL Offs(pOrigin,262.28,51.59,0.00),v60,z0,tPen\WObj:=wPaper;
    MoveL Offs(pOrigin,264.53,49.34,0.00),v40,fine,tPen\WObj:=wPaper;
    MoveL Offs(pOrigin,264.53,49.34,6.00),v60,z5,tPen\WObj:=wPaper;
    MoveL Offs(pOrigin,266.47,50.38,6.00),vTravel,z5,tPen\WObj:=wPaper;
    MoveL Offs(pOrigin,266.47,50.38,0.00),v60,z0,tPen\WObj:=wPaper;
    MoveL Offs(pOrigin,264.22,52.63,0.00),v40,z0,tPen\WObj:=wPaper;
    MoveL Offs(pOrigin,265.12,53.23,0.00),v40,z0,tPen\WObj:=wPaper;
    MoveL Offs(pOrigin,267.37,50.98,0.00),v40,fine,tPen\WObj:=wPaper;
    MoveL Offs(pOrigin,267.37,50.98,6.00),v60,z5,tPen\WObj:=wPaper;
    MoveL Offs(pOrigin,268.06,49.20,6.00),vTravel,z5,tPen\WObj:=wPaper;
    MoveL Offs(pOrigin,268.06,49.20,0.00),v60,z0,tPen\WObj:=wPaper;
    MoveL Offs(pOrigin,269.62,47.08,0.00),v40,z0,tPen\WObj:=wPaper;
    MoveL Offs(pOrigin,269.76,46.22,0.00),v40,fine,tPen\WObj:=wPaper;
    MoveL Offs(pOrigin,269.76,46.22,6.00),v60,z5,tPen\WObj:=wPaper;
    MoveL Offs(pOrigin,271.74,43.62,6.00),vTravel,z5,tPen\WObj:=wPaper;
    MoveL Offs(pOrigin,271.74,43.62,0.00),v60,z0,tPen\WObj:=wPaper;
    MoveL Offs(pOrigin,273.99,41.37,0.00),v40,z0,tPen\WObj:=wPaper;
    MoveL Offs(pOrigin,273.09,40.77,0.00),v40,z0,tPen\WObj:=wPaper;
    MoveL Offs(pOrigin,270.84,43.03,0.00),v40,fine,tPen\WObj:=wPaper;
    MoveL Offs(pOrigin,270.84,43.03,6.00),v60,z5,tPen\WObj:=wPaper;
    MoveL Offs(pOrigin,272.31,42.46,6.00),vTravel,z5,tPen\WObj:=wPaper;
  ENDPROC

  PROC DrawPart87()
    MoveL Offs(pOrigin,272.31,42.46,0.00),v60,z0,tPen\WObj:=wPaper;
    MoveL Offs(pOrigin,274.01,42.46,0.00),v40,fine,tPen\WObj:=wPaper;
    MoveL Offs(pOrigin,274.01,42.46,6.00),v60,z5,tPen\WObj:=wPaper;
    MoveL Offs(pOrigin,275.04,41.81,6.00),vTravel,z5,tPen\WObj:=wPaper;
    MoveL Offs(pOrigin,275.04,41.81,0.00),v60,z0,tPen\WObj:=wPaper;
    MoveL Offs(pOrigin,272.93,43.92,0.00),v40,fine,tPen\WObj:=wPaper;
    MoveL Offs(pOrigin,272.93,43.92,6.00),v60,z5,tPen\WObj:=wPaper;
    MoveL Offs(pOrigin,274.65,43.51,6.00),vTravel,z5,tPen\WObj:=wPaper;
    MoveL Offs(pOrigin,274.65,43.51,0.00),v60,z0,tPen\WObj:=wPaper;
    MoveL Offs(pOrigin,276.35,43.51,0.00),v40,z0,tPen\WObj:=wPaper;
    MoveL Offs(pOrigin,277.13,42.71,0.00),v40,z0,tPen\WObj:=wPaper;
    MoveL Offs(pOrigin,274.88,44.96,0.00),v40,fine,tPen\WObj:=wPaper;
    MoveL Offs(pOrigin,274.88,44.96,6.00),v60,z5,tPen\WObj:=wPaper;
    MoveL Offs(pOrigin,276.99,44.57,6.00),vTravel,z5,tPen\WObj:=wPaper;
    MoveL Offs(pOrigin,276.99,44.57,0.00),v60,z0,tPen\WObj:=wPaper;
    MoveL Offs(pOrigin,278.90,44.57,0.00),v40,z0,tPen\WObj:=wPaper;
    MoveL Offs(pOrigin,279.23,43.60,0.00),v40,z0,tPen\WObj:=wPaper;
    MoveL Offs(pOrigin,276.82,46.00,0.00),v40,z0,tPen\WObj:=wPaper;
    MoveL Offs(pOrigin,277.87,46.45,0.00),v40,z0,tPen\WObj:=wPaper;
    MoveL Offs(pOrigin,280.27,44.04,0.00),v40,fine,tPen\WObj:=wPaper;
    MoveL Offs(pOrigin,280.27,44.04,6.00),v60,z5,tPen\WObj:=wPaper;
    MoveL Offs(pOrigin,279.96,45.62,6.00),vTravel,z5,tPen\WObj:=wPaper;
    MoveL Offs(pOrigin,279.96,45.62,0.00),v60,z0,tPen\WObj:=wPaper;
    MoveL Offs(pOrigin,286.98,45.62,0.00),v40,z0,tPen\WObj:=wPaper;
    MoveL Offs(pOrigin,286.12,46.01,0.00),v40,z0,tPen\WObj:=wPaper;
    MoveL Offs(pOrigin,286.34,46.65,0.00),v40,z0,tPen\WObj:=wPaper;
    MoveL Offs(pOrigin,286.76,46.86,0.00),v40,z0,tPen\WObj:=wPaper;
    MoveL Offs(pOrigin,286.98,46.68,0.00),v40,z0,tPen\WObj:=wPaper;
    MoveL Offs(pOrigin,282.94,46.68,0.00),v40,fine,tPen\WObj:=wPaper;
    MoveL Offs(pOrigin,282.94,46.68,6.00),v60,z5,tPen\WObj:=wPaper;
    MoveL Offs(pOrigin,282.36,47.93,6.00),vTravel,z5,tPen\WObj:=wPaper;
    MoveL Offs(pOrigin,282.36,47.93,0.00),v60,z0,tPen\WObj:=wPaper;
    MoveL Offs(pOrigin,293.78,36.51,0.00),v40,z0,tPen\WObj:=wPaper;
    MoveL Offs(pOrigin,292.73,36.07,0.00),v40,z0,tPen\WObj:=wPaper;
    MoveL Offs(pOrigin,281.31,47.49,0.00),v40,fine,tPen\WObj:=wPaper;
    MoveL Offs(pOrigin,281.31,47.49,6.00),v60,z5,tPen\WObj:=wPaper;
    MoveL Offs(pOrigin,286.12,46.01,6.00),vTravel,z5,tPen\WObj:=wPaper;
    MoveL Offs(pOrigin,286.12,46.01,0.00),v60,z0,tPen\WObj:=wPaper;
    MoveL Offs(pOrigin,286.76,45.59,0.00),v40,z0,tPen\WObj:=wPaper;
    MoveL Offs(pOrigin,289.31,45.80,0.00),v40,z0,tPen\WObj:=wPaper;
    MoveL Offs(pOrigin,289.36,46.23,0.00),v40,z0,tPen\WObj:=wPaper;
    MoveL Offs(pOrigin,287.41,44.28,0.00),v40,z0,tPen\WObj:=wPaper;
    MoveL Offs(pOrigin,288.46,43.83,0.00),v40,z0,tPen\WObj:=wPaper;
    MoveL Offs(pOrigin,290.11,45.48,0.00),v40,fine,tPen\WObj:=wPaper;
    MoveL Offs(pOrigin,290.11,45.48,6.00),v60,z5,tPen\WObj:=wPaper;
    MoveL Offs(pOrigin,289.52,44.31,6.00),vTravel,z5,tPen\WObj:=wPaper;
    MoveL Offs(pOrigin,289.52,44.31,0.00),v60,z0,tPen\WObj:=wPaper;
    MoveL Offs(pOrigin,289.74,42.83,0.00),v40,z0,tPen\WObj:=wPaper;
    MoveL Offs(pOrigin,289.74,42.83,0.00),v40,z0,tPen\WObj:=wPaper;
    MoveL Offs(pOrigin,286.98,41.34,0.00),v40,z0,tPen\WObj:=wPaper;
    MoveL Offs(pOrigin,286.98,41.34,0.00),v40,z0,tPen\WObj:=wPaper;
    MoveL Offs(pOrigin,287.61,41.97,0.00),v40,fine,tPen\WObj:=wPaper;
    MoveL Offs(pOrigin,287.61,41.97,6.00),v60,z5,tPen\WObj:=wPaper;
    MoveL Offs(pOrigin,289.35,41.74,6.00),vTravel,z5,tPen\WObj:=wPaper;
    MoveL Offs(pOrigin,289.35,41.74,0.00),v60,z0,tPen\WObj:=wPaper;
    MoveL Offs(pOrigin,291.00,43.39,0.00),v40,fine,tPen\WObj:=wPaper;
    MoveL Offs(pOrigin,291.00,43.39,6.00),v60,z5,tPen\WObj:=wPaper;
    MoveL Offs(pOrigin,288.47,46.83,6.00),vTravel,z5,tPen\WObj:=wPaper;
    MoveL Offs(pOrigin,288.47,46.83,0.00),v60,z0,tPen\WObj:=wPaper;
    MoveL Offs(pOrigin,283.96,42.32,0.00),v40,fine,tPen\WObj:=wPaper;
    MoveL Offs(pOrigin,283.96,42.32,6.00),v60,z5,tPen\WObj:=wPaper;
    MoveL Offs(pOrigin,285.70,36.12,6.00),vTravel,z5,tPen\WObj:=wPaper;
    MoveL Offs(pOrigin,285.70,36.12,0.00),v60,z0,tPen\WObj:=wPaper;
    MoveL Offs(pOrigin,290.16,36.12,0.00),v40,fine,tPen\WObj:=wPaper;
    MoveL Offs(pOrigin,290.16,36.12,6.00),v60,z5,tPen\WObj:=wPaper;
    MoveL Offs(pOrigin,289.52,37.30,6.00),vTravel,z5,tPen\WObj:=wPaper;
    MoveL Offs(pOrigin,289.52,37.30,0.00),v60,z0,tPen\WObj:=wPaper;
    MoveL Offs(pOrigin,289.74,37.72,0.00),v40,z0,tPen\WObj:=wPaper;
    MoveL Offs(pOrigin,289.52,37.30,0.00),v40,z0,tPen\WObj:=wPaper;
    MoveL Offs(pOrigin,288.68,37.18,0.00),v40,z0,tPen\WObj:=wPaper;
    MoveL Offs(pOrigin,292.29,37.18,0.00),v40,fine,tPen\WObj:=wPaper;
    MoveL Offs(pOrigin,292.29,37.18,6.00),v60,z5,tPen\WObj:=wPaper;
    MoveL Offs(pOrigin,291.65,38.23,6.00),vTravel,z5,tPen\WObj:=wPaper;
    MoveL Offs(pOrigin,291.65,38.23,0.00),v60,z0,tPen\WObj:=wPaper;
    MoveL Offs(pOrigin,290.59,38.23,0.00),v40,z0,tPen\WObj:=wPaper;
    MoveL Offs(pOrigin,291.01,38.36,0.00),v40,z0,tPen\WObj:=wPaper;
    MoveL Offs(pOrigin,289.95,38.36,0.00),v40,fine,tPen\WObj:=wPaper;
    MoveL Offs(pOrigin,289.95,38.36,6.00),v60,z5,tPen\WObj:=wPaper;
    MoveL Offs(pOrigin,285.49,35.81,6.00),vTravel,z5,tPen\WObj:=wPaper;
    MoveL Offs(pOrigin,285.49,35.81,0.00),v60,z0,tPen\WObj:=wPaper;
    MoveL Offs(pOrigin,285.70,36.24,0.00),v40,z0,tPen\WObj:=wPaper;
    MoveL Offs(pOrigin,285.49,35.81,0.00),v40,fine,tPen\WObj:=wPaper;
    MoveL Offs(pOrigin,285.49,35.81,6.00),v60,z5,tPen\WObj:=wPaper;
    MoveL Offs(pOrigin,285.06,34.01,6.00),vTravel,z5,tPen\WObj:=wPaper;
    MoveL Offs(pOrigin,285.06,34.01,0.00),v60,z0,tPen\WObj:=wPaper;
    MoveL Offs(pOrigin,282.94,34.01,0.00),v40,z0,tPen\WObj:=wPaper;
    MoveL Offs(pOrigin,282.51,32.95,0.00),v40,z0,tPen\WObj:=wPaper;
    MoveL Offs(pOrigin,280.18,32.95,0.00),v40,z0,tPen\WObj:=wPaper;
    MoveL Offs(pOrigin,279.96,31.90,0.00),v40,z0,tPen\WObj:=wPaper;
    MoveL Offs(pOrigin,277.20,31.90,0.00),v40,fine,tPen\WObj:=wPaper;
    MoveL Offs(pOrigin,277.20,31.90,6.00),v60,z5,tPen\WObj:=wPaper;
    MoveL Offs(pOrigin,277.61,33.27,6.00),vTravel,z5,tPen\WObj:=wPaper;
    MoveL Offs(pOrigin,277.61,33.27,0.00),v60,z0,tPen\WObj:=wPaper;
    MoveL Offs(pOrigin,280.01,30.86,0.00),v40,z0,tPen\WObj:=wPaper;
    MoveL Offs(pOrigin,281.06,31.31,0.00),v40,z0,tPen\WObj:=wPaper;
    MoveL Offs(pOrigin,278.66,33.71,0.00),v40,fine,tPen\WObj:=wPaper;
    MoveL Offs(pOrigin,278.66,33.71,6.00),v60,z5,tPen\WObj:=wPaper;
    MoveL Offs(pOrigin,280.90,34.46,6.00),vTravel,z5,tPen\WObj:=wPaper;
    MoveL Offs(pOrigin,280.90,34.46,0.00),v60,z0,tPen\WObj:=wPaper;
    MoveL Offs(pOrigin,283.31,32.05,0.00),v40,fine,tPen\WObj:=wPaper;
    MoveL Offs(pOrigin,283.31,32.05,6.00),v60,z5,tPen\WObj:=wPaper;
    MoveL Offs(pOrigin,284.42,33.69,6.00),vTravel,z5,tPen\WObj:=wPaper;
    MoveL Offs(pOrigin,284.42,33.69,0.00),v60,z0,tPen\WObj:=wPaper;
    MoveL Offs(pOrigin,284.85,33.90,0.00),v40,z0,tPen\WObj:=wPaper;
    MoveL Offs(pOrigin,284.42,33.69,0.00),v40,fine,tPen\WObj:=wPaper;
    MoveL Offs(pOrigin,284.42,33.69,6.00),v60,z5,tPen\WObj:=wPaper;
    MoveL Offs(pOrigin,285.40,32.94,6.00),vTravel,z5,tPen\WObj:=wPaper;
    MoveL Offs(pOrigin,285.40,32.94,0.00),v60,z0,tPen\WObj:=wPaper;
    MoveL Offs(pOrigin,283.00,35.35,0.00),v40,fine,tPen\WObj:=wPaper;
    MoveL Offs(pOrigin,283.00,35.35,6.00),v60,z5,tPen\WObj:=wPaper;
    MoveL Offs(pOrigin,277.20,36.24,6.00),vTravel,z5,tPen\WObj:=wPaper;
    MoveL Offs(pOrigin,277.20,36.24,0.00),v60,z0,tPen\WObj:=wPaper;
    MoveL Offs(pOrigin,276.35,37.72,0.00),v40,z0,tPen\WObj:=wPaper;
    MoveL Offs(pOrigin,276.35,38.36,0.00),v40,fine,tPen\WObj:=wPaper;
    MoveL Offs(pOrigin,276.35,38.36,6.00),v60,z5,tPen\WObj:=wPaper;
    MoveL Offs(pOrigin,275.52,32.38,6.00),vTravel,z5,tPen\WObj:=wPaper;
    MoveL Offs(pOrigin,275.52,32.38,0.00),v60,z0,tPen\WObj:=wPaper;
    MoveL Offs(pOrigin,277.77,30.12,0.00),v40,fine,tPen\WObj:=wPaper;
    MoveL Offs(pOrigin,277.77,30.12,6.00),v60,z5,tPen\WObj:=wPaper;
    MoveL Offs(pOrigin,276.57,29.83,6.00),vTravel,z5,tPen\WObj:=wPaper;
  ENDPROC

  PROC DrawPart88()
    MoveL Offs(pOrigin,276.57,29.83,0.00),v60,z0,tPen\WObj:=wPaper;
    MoveL Offs(pOrigin,274.17,32.23,0.00),v40,z0,tPen\WObj:=wPaper;
    MoveL Offs(pOrigin,274.79,31.66,0.00),v40,z0,tPen\WObj:=wPaper;
    MoveL Offs(pOrigin,265.77,22.64,0.00),v40,fine,tPen\WObj:=wPaper;
    MoveL Offs(pOrigin,265.77,22.64,6.00),v60,z5,tPen\WObj:=wPaper;
    MoveL Offs(pOrigin,262.54,24.50,6.00),vTravel,z5,tPen\WObj:=wPaper;
    MoveL Offs(pOrigin,262.54,24.50,0.00),v60,z0,tPen\WObj:=wPaper;
    MoveL Offs(pOrigin,259.99,24.50,0.00),v40,fine,tPen\WObj:=wPaper;
    MoveL Offs(pOrigin,259.99,24.50,6.00),v60,z5,tPen\WObj:=wPaper;
    MoveL Offs(pOrigin,258.08,23.45,6.00),vTravel,z5,tPen\WObj:=wPaper;
    MoveL Offs(pOrigin,258.08,23.45,0.00),v60,z0,tPen\WObj:=wPaper;
    MoveL Offs(pOrigin,255.52,23.45,0.00),v40,z0,tPen\WObj:=wPaper;
    MoveL Offs(pOrigin,255.29,24.11,0.00),v40,z0,tPen\WObj:=wPaper;
    MoveL Offs(pOrigin,249.88,18.70,0.00),v40,fine,tPen\WObj:=wPaper;
    MoveL Offs(pOrigin,249.88,18.70,6.00),v60,z5,tPen\WObj:=wPaper;
    MoveL Offs(pOrigin,251.27,19.24,6.00),vTravel,z5,tPen\WObj:=wPaper;
    MoveL Offs(pOrigin,251.27,19.24,0.00),v60,z0,tPen\WObj:=wPaper;
    MoveL Offs(pOrigin,256.80,20.73,0.00),v40,z0,tPen\WObj:=wPaper;
    MoveL Offs(pOrigin,256.80,21.36,0.00),v40,z0,tPen\WObj:=wPaper;
    MoveL Offs(pOrigin,251.27,19.88,0.00),v40,fine,tPen\WObj:=wPaper;
    MoveL Offs(pOrigin,251.27,19.88,6.00),v60,z5,tPen\WObj:=wPaper;
    MoveL Offs(pOrigin,250.00,21.34,6.00),vTravel,z5,tPen\WObj:=wPaper;
    MoveL Offs(pOrigin,250.00,21.34,0.00),v60,z0,tPen\WObj:=wPaper;
    MoveL Offs(pOrigin,247.02,21.34,0.00),v40,z0,tPen\WObj:=wPaper;
    MoveL Offs(pOrigin,247.35,22.13,0.00),v40,z0,tPen\WObj:=wPaper;
    MoveL Offs(pOrigin,241.34,16.12,0.00),v40,fine,tPen\WObj:=wPaper;
    MoveL Offs(pOrigin,241.34,16.12,6.00),v60,z5,tPen\WObj:=wPaper;
    MoveL Offs(pOrigin,241.92,19.22,6.00),vTravel,z5,tPen\WObj:=wPaper;
    MoveL Offs(pOrigin,241.92,19.22,0.00),v60,z0,tPen\WObj:=wPaper;
    MoveL Offs(pOrigin,238.31,19.22,0.00),v40,z0,tPen\WObj:=wPaper;
    MoveL Offs(pOrigin,237.30,19.56,0.00),v40,z0,tPen\WObj:=wPaper;
    MoveL Offs(pOrigin,234.90,17.15,0.00),v40,z0,tPen\WObj:=wPaper;
    MoveL Offs(pOrigin,235.64,16.41,0.00),v40,z0,tPen\WObj:=wPaper;
    MoveL Offs(pOrigin,230.69,11.45,0.00),v40,fine,tPen\WObj:=wPaper;
    MoveL Offs(pOrigin,230.69,11.45,6.00),v60,z5,tPen\WObj:=wPaper;
    MoveL Offs(pOrigin,228.25,10.95,6.00),vTravel,z5,tPen\WObj:=wPaper;
    MoveL Offs(pOrigin,228.25,10.95,0.00),v60,z0,tPen\WObj:=wPaper;
    MoveL Offs(pOrigin,216.22,22.97,0.00),v40,z0,tPen\WObj:=wPaper;
    MoveL Offs(pOrigin,216.49,22.64,0.00),v40,z0,tPen\WObj:=wPaper;
    MoveL Offs(pOrigin,212.88,19.03,0.00),v40,z0,tPen\WObj:=wPaper;
    MoveL Offs(pOrigin,212.27,19.88,0.00),v40,z0,tPen\WObj:=wPaper;
    MoveL Offs(pOrigin,212.27,21.15,0.00),v40,z0,tPen\WObj:=wPaper;
    MoveL Offs(pOrigin,211.54,21.79,0.00),v40,z0,tPen\WObj:=wPaper;
    MoveL Offs(pOrigin,212.81,21.58,0.00),v40,z0,tPen\WObj:=wPaper;
    MoveL Offs(pOrigin,238.74,27.31,0.00),v40,z0,tPen\WObj:=wPaper;
    MoveL Offs(pOrigin,245.75,28.59,0.00),v40,fine,tPen\WObj:=wPaper;
    MoveL Offs(pOrigin,245.75,28.59,6.00),v60,z5,tPen\WObj:=wPaper;
    MoveL Offs(pOrigin,241.38,26.19,6.00),vTravel,z5,tPen\WObj:=wPaper;
    MoveL Offs(pOrigin,241.38,26.19,0.00),v60,z0,tPen\WObj:=wPaper;
    MoveL Offs(pOrigin,239.43,28.14,0.00),v40,z0,tPen\WObj:=wPaper;
    MoveL Offs(pOrigin,239.42,27.65,0.00),v40,z0,tPen\WObj:=wPaper;
    MoveL Offs(pOrigin,237.77,26.00,0.00),v40,z0,tPen\WObj:=wPaper;
    MoveL Offs(pOrigin,237.79,25.30,0.00),v40,z0,tPen\WObj:=wPaper;
    MoveL Offs(pOrigin,235.84,27.25,0.00),v40,z0,tPen\WObj:=wPaper;
    MoveL Offs(pOrigin,235.83,27.04,0.00),v40,z0,tPen\WObj:=wPaper;
    MoveL Offs(pOrigin,234.02,25.24,0.00),v40,z0,tPen\WObj:=wPaper;
    MoveL Offs(pOrigin,234.05,24.56,0.00),v40,z0,tPen\WObj:=wPaper;
    MoveL Offs(pOrigin,232.09,26.52,0.00),v40,z0,tPen\WObj:=wPaper;
    MoveL Offs(pOrigin,231.93,26.13,0.00),v40,z0,tPen\WObj:=wPaper;
    MoveL Offs(pOrigin,230.13,24.33,0.00),v40,z0,tPen\WObj:=wPaper;
    MoveL Offs(pOrigin,230.30,23.83,0.00),v40,z0,tPen\WObj:=wPaper;
    MoveL Offs(pOrigin,228.35,25.78,0.00),v40,z0,tPen\WObj:=wPaper;
    MoveL Offs(pOrigin,228.03,25.22,0.00),v40,z0,tPen\WObj:=wPaper;
    MoveL Offs(pOrigin,226.23,23.42,0.00),v40,z0,tPen\WObj:=wPaper;
    MoveL Offs(pOrigin,226.71,22.94,0.00),v40,z0,tPen\WObj:=wPaper;
    MoveL Offs(pOrigin,224.76,24.89,0.00),v40,z0,tPen\WObj:=wPaper;
    MoveL Offs(pOrigin,224.28,24.46,0.00),v40,z0,tPen\WObj:=wPaper;
    MoveL Offs(pOrigin,222.63,22.81,0.00),v40,z0,tPen\WObj:=wPaper;
    MoveL Offs(pOrigin,223.12,22.05,0.00),v40,z0,tPen\WObj:=wPaper;
    MoveL Offs(pOrigin,221.16,24.00,0.00),v40,z0,tPen\WObj:=wPaper;
    MoveL Offs(pOrigin,220.39,23.55,0.00),v40,z0,tPen\WObj:=wPaper;
    MoveL Offs(pOrigin,218.58,21.75,0.00),v40,z0,tPen\WObj:=wPaper;
    MoveL Offs(pOrigin,219.53,21.16,0.00),v40,z0,tPen\WObj:=wPaper;
    MoveL Offs(pOrigin,217.27,23.42,0.00),v40,fine,tPen\WObj:=wPaper;
    MoveL Offs(pOrigin,217.27,23.42,6.00),v60,z5,tPen\WObj:=wPaper;
    MoveL Offs(pOrigin,214.88,22.82,6.00),vTravel,z5,tPen\WObj:=wPaper;
    MoveL Offs(pOrigin,214.88,22.82,0.00),v60,z0,tPen\WObj:=wPaper;
    MoveL Offs(pOrigin,226.75,10.95,0.00),v40,fine,tPen\WObj:=wPaper;
    MoveL Offs(pOrigin,226.75,10.95,6.00),v60,z5,tPen\WObj:=wPaper;
    MoveL Offs(pOrigin,227.84,11.59,6.00),vTravel,z5,tPen\WObj:=wPaper;
    MoveL Offs(pOrigin,227.84,11.59,0.00),v60,z0,tPen\WObj:=wPaper;
    MoveL Offs(pOrigin,232.05,15.80,0.00),v40,fine,tPen\WObj:=wPaper;
    MoveL Offs(pOrigin,232.05,15.80,6.00),v60,z5,tPen\WObj:=wPaper;
    MoveL Offs(pOrigin,231.90,17.14,6.00),vTravel,z5,tPen\WObj:=wPaper;
    MoveL Offs(pOrigin,231.90,17.14,0.00),v60,z0,tPen\WObj:=wPaper;
    MoveL Offs(pOrigin,233.70,18.95,0.00),v40,z0,tPen\WObj:=wPaper;
    MoveL Offs(pOrigin,233.31,19.32,0.00),v40,z0,tPen\WObj:=wPaper;
    MoveL Offs(pOrigin,240.38,12.26,0.00),v40,z0,tPen\WObj:=wPaper;
    MoveL Offs(pOrigin,240.44,12.89,0.00),v40,z0,tPen\WObj:=wPaper;
    MoveL Offs(pOrigin,217.06,12.89,0.00),v40,z0,tPen\WObj:=wPaper;
    MoveL Offs(pOrigin,217.21,12.90,0.00),v40,z0,tPen\WObj:=wPaper;
    MoveL Offs(pOrigin,221.12,16.81,0.00),v40,fine,tPen\WObj:=wPaper;
    MoveL Offs(pOrigin,221.12,16.81,6.00),v60,z5,tPen\WObj:=wPaper;
    MoveL Offs(pOrigin,219.77,16.96,6.00),vTravel,z5,tPen\WObj:=wPaper;
    MoveL Offs(pOrigin,219.77,16.96,0.00),v60,z0,tPen\WObj:=wPaper;
    MoveL Offs(pOrigin,215.71,12.90,0.00),v40,z0,tPen\WObj:=wPaper;
    MoveL Offs(pOrigin,216.41,12.33,0.00),v40,z0,tPen\WObj:=wPaper;
    MoveL Offs(pOrigin,205.29,23.45,0.00),v40,z0,tPen\WObj:=wPaper;
    MoveL Offs(pOrigin,205.11,23.20,0.00),v40,z0,tPen\WObj:=wPaper;
    MoveL Offs(pOrigin,203.15,21.25,0.00),v40,z0,tPen\WObj:=wPaper;
    MoveL Offs(pOrigin,203.80,20.46,0.00),v40,z0,tPen\WObj:=wPaper;
    MoveL Offs(pOrigin,200.19,24.07,0.00),v40,z0,tPen\WObj:=wPaper;
    MoveL Offs(pOrigin,199.72,23.79,0.00),v40,z0,tPen\WObj:=wPaper;
    MoveL Offs(pOrigin,197.61,21.68,0.00),v40,z0,tPen\WObj:=wPaper;
    MoveL Offs(pOrigin,197.51,21.58,0.00),v40,z0,tPen\WObj:=wPaper;
    MoveL Offs(pOrigin,196.88,21.58,0.00),v40,z0,tPen\WObj:=wPaper;
    MoveL Offs(pOrigin,196.45,21.15,0.00),v40,z0,tPen\WObj:=wPaper;
    MoveL Offs(pOrigin,196.24,21.34,0.00),v40,z0,tPen\WObj:=wPaper;
    MoveL Offs(pOrigin,193.26,21.34,0.00),v40,z0,tPen\WObj:=wPaper;
    MoveL Offs(pOrigin,192.52,21.07,0.00),v40,z0,tPen\WObj:=wPaper;
    MoveL Offs(pOrigin,194.47,23.02,0.00),v40,z0,tPen\WObj:=wPaper;
    MoveL Offs(pOrigin,194.80,23.49,0.00),v40,z0,tPen\WObj:=wPaper;
    MoveL Offs(pOrigin,197.66,20.63,0.00),v40,z0,tPen\WObj:=wPaper;
    MoveL Offs(pOrigin,197.06,19.73,0.00),v40,z0,tPen\WObj:=wPaper;
    MoveL Offs(pOrigin,193.60,23.19,0.00),v40,z0,tPen\WObj:=wPaper;
    MoveL Offs(pOrigin,192.67,22.72,0.00),v40,z0,tPen\WObj:=wPaper;
    MoveL Offs(pOrigin,191.47,21.51,0.00),v40,fine,tPen\WObj:=wPaper;
    MoveL Offs(pOrigin,191.47,21.51,6.00),v60,z5,tPen\WObj:=wPaper;
    MoveL Offs(pOrigin,190.12,21.66,6.00),vTravel,z5,tPen\WObj:=wPaper;
    MoveL Offs(pOrigin,190.12,21.66,0.00),v60,z0,tPen\WObj:=wPaper;
  ENDPROC

  PROC DrawPart89()
    MoveL Offs(pOrigin,191.47,23.01,0.00),v40,z0,tPen\WObj:=wPaper;
    MoveL Offs(pOrigin,191.81,23.49,0.00),v40,z0,tPen\WObj:=wPaper;
    MoveL Offs(pOrigin,196.91,18.39,0.00),v40,z0,tPen\WObj:=wPaper;
    MoveL Offs(pOrigin,195.80,18.38,0.00),v40,z0,tPen\WObj:=wPaper;
    MoveL Offs(pOrigin,192.65,15.23,0.00),v40,z0,tPen\WObj:=wPaper;
    MoveL Offs(pOrigin,193.26,15.84,0.00),v40,z0,tPen\WObj:=wPaper;
    MoveL Offs(pOrigin,193.26,19.66,0.00),v40,z0,tPen\WObj:=wPaper;
    MoveL Offs(pOrigin,193.26,20.28,0.00),v40,z0,tPen\WObj:=wPaper;
    MoveL Offs(pOrigin,195.18,20.28,0.00),v40,z0,tPen\WObj:=wPaper;
    MoveL Offs(pOrigin,195.96,20.03,0.00),v40,z0,tPen\WObj:=wPaper;
    MoveL Offs(pOrigin,191.45,15.52,0.00),v40,z0,tPen\WObj:=wPaper;
    MoveL Offs(pOrigin,191.68,14.66,0.00),v40,z0,tPen\WObj:=wPaper;
    MoveL Offs(pOrigin,181.92,24.42,0.00),v40,z0,tPen\WObj:=wPaper;
    MoveL Offs(pOrigin,181.74,23.73,0.00),v40,z0,tPen\WObj:=wPaper;
    MoveL Offs(pOrigin,180.69,22.68,0.00),v40,z0,tPen\WObj:=wPaper;
    MoveL Offs(pOrigin,180.24,23.73,0.00),v40,z0,tPen\WObj:=wPaper;
    MoveL Offs(pOrigin,179.34,22.82,0.00),v40,fine,tPen\WObj:=wPaper;
    MoveL Offs(pOrigin,179.34,22.82,6.00),v60,z5,tPen\WObj:=wPaper;
    MoveL Offs(pOrigin,179.04,24.02,6.00),vTravel,z5,tPen\WObj:=wPaper;
    MoveL Offs(pOrigin,179.04,24.02,0.00),v60,z0,tPen\WObj:=wPaper;
    MoveL Offs(pOrigin,177.84,22.82,0.00),v40,fine,tPen\WObj:=wPaper;
    MoveL Offs(pOrigin,177.84,22.82,6.00),v60,z5,tPen\WObj:=wPaper;
    MoveL Offs(pOrigin,176.64,23.12,6.00),vTravel,z5,tPen\WObj:=wPaper;
    MoveL Offs(pOrigin,176.64,23.12,0.00),v60,z0,tPen\WObj:=wPaper;
    MoveL Offs(pOrigin,177.70,24.17,0.00),v40,z0,tPen\WObj:=wPaper;
    MoveL Offs(pOrigin,177.12,24.74,0.00),v40,z0,tPen\WObj:=wPaper;
    MoveL Offs(pOrigin,186.44,15.42,0.00),v40,z0,tPen\WObj:=wPaper;
    MoveL Offs(pOrigin,186.25,16.06,0.00),v40,z0,tPen\WObj:=wPaper;
    MoveL Offs(pOrigin,196.02,16.06,0.00),v40,fine,tPen\WObj:=wPaper;
    MoveL Offs(pOrigin,196.02,16.06,6.00),v60,z5,tPen\WObj:=wPaper;
    MoveL Offs(pOrigin,196.09,14.19,6.00),vTravel,z5,tPen\WObj:=wPaper;
    MoveL Offs(pOrigin,196.09,14.19,0.00),v60,z0,tPen\WObj:=wPaper;
    MoveL Offs(pOrigin,198.34,16.44,0.00),v40,z0,tPen\WObj:=wPaper;
    MoveL Offs(pOrigin,198.42,16.88,0.00),v40,z0,tPen\WObj:=wPaper;
    MoveL Offs(pOrigin,202.47,12.83,0.00),v40,z0,tPen\WObj:=wPaper;
    MoveL Offs(pOrigin,202.83,13.46,0.00),v40,z0,tPen\WObj:=wPaper;
    MoveL Offs(pOrigin,211.54,22.17,0.00),v40,z0,tPen\WObj:=wPaper;
    MoveL Offs(pOrigin,210.90,22.00,0.00),v40,z0,tPen\WObj:=wPaper;
    MoveL Offs(pOrigin,209.84,22.42,0.00),v40,z0,tPen\WObj:=wPaper;
    MoveL Offs(pOrigin,199.43,23.49,0.00),v40,z0,tPen\WObj:=wPaper;
    MoveL Offs(pOrigin,196.66,23.49,0.00),v40,z0,tPen\WObj:=wPaper;
    MoveL Offs(pOrigin,194.54,22.42,0.00),v40,z0,tPen\WObj:=wPaper;
    MoveL Offs(pOrigin,129.94,28.38,0.00),v40,z0,tPen\WObj:=wPaper;
    MoveL Offs(pOrigin,129.62,28.36,0.00),v40,z0,tPen\WObj:=wPaper;
    MoveL Offs(pOrigin,126.47,25.21,0.00),v40,z0,tPen\WObj:=wPaper;
    MoveL Offs(pOrigin,125.72,24.46,0.00),v40,z0,tPen\WObj:=wPaper;
    MoveL Offs(pOrigin,123.91,22.65,0.00),v40,fine,tPen\WObj:=wPaper;
    MoveL Offs(pOrigin,123.91,22.65,6.00),v60,z5,tPen\WObj:=wPaper;
    MoveL Offs(pOrigin,128.66,22.39,6.00),vTravel,z5,tPen\WObj:=wPaper;
    MoveL Offs(pOrigin,128.66,22.39,0.00),v60,z0,tPen\WObj:=wPaper;
    MoveL Offs(pOrigin,139.29,22.39,0.00),v40,z0,tPen\WObj:=wPaper;
    MoveL Offs(pOrigin,139.19,23.00,0.00),v40,z0,tPen\WObj:=wPaper;
    MoveL Offs(pOrigin,137.39,21.20,0.00),v40,z0,tPen\WObj:=wPaper;
    MoveL Offs(pOrigin,138.04,20.51,0.00),v40,z0,tPen\WObj:=wPaper;
    MoveL Offs(pOrigin,129.47,29.08,0.00),v40,fine,tPen\WObj:=wPaper;
    MoveL Offs(pOrigin,129.47,29.08,6.00),v60,z5,tPen\WObj:=wPaper;
    MoveL Offs(pOrigin,129.94,27.10,6.00),vTravel,z5,tPen\WObj:=wPaper;
    MoveL Offs(pOrigin,129.94,27.10,0.00),v60,z0,tPen\WObj:=wPaper;
    MoveL Offs(pOrigin,131.43,26.67,0.00),v40,z0,tPen\WObj:=wPaper;
    MoveL Offs(pOrigin,132.70,27.10,0.00),v40,z0,tPen\WObj:=wPaper;
    MoveL Offs(pOrigin,133.98,26.75,0.00),v40,z0,tPen\WObj:=wPaper;
    MoveL Offs(pOrigin,135.46,27.10,0.00),v40,z0,tPen\WObj:=wPaper;
    MoveL Offs(pOrigin,136.10,26.25,0.00),v40,z0,tPen\WObj:=wPaper;
    MoveL Offs(pOrigin,134.61,26.04,0.00),v40,z0,tPen\WObj:=wPaper;
    MoveL Offs(pOrigin,134.33,26.25,0.00),v40,z0,tPen\WObj:=wPaper;
    MoveL Offs(pOrigin,134.61,26.89,0.00),v40,z0,tPen\WObj:=wPaper;
    MoveL Offs(pOrigin,135.01,27.78,0.00),v40,z0,tPen\WObj:=wPaper;
    MoveL Offs(pOrigin,131.86,24.63,0.00),v40,z0,tPen\WObj:=wPaper;
    MoveL Offs(pOrigin,132.46,23.73,0.00),v40,z0,tPen\WObj:=wPaper;
    MoveL Offs(pOrigin,130.80,22.08,0.00),v40,fine,tPen\WObj:=wPaper;
    MoveL Offs(pOrigin,130.80,22.08,6.00),v60,z5,tPen\WObj:=wPaper;
    MoveL Offs(pOrigin,133.55,25.83,6.00),vTravel,z5,tPen\WObj:=wPaper;
    MoveL Offs(pOrigin,133.55,25.83,0.00),v60,z0,tPen\WObj:=wPaper;
    MoveL Offs(pOrigin,133.90,26.32,0.00),v40,z0,tPen\WObj:=wPaper;
    MoveL Offs(pOrigin,132.91,25.83,0.00),v40,z0,tPen\WObj:=wPaper;
    MoveL Offs(pOrigin,132.06,26.67,0.00),v40,fine,tPen\WObj:=wPaper;
    MoveL Offs(pOrigin,132.06,26.67,6.00),v60,z5,tPen\WObj:=wPaper;
    MoveL Offs(pOrigin,136.38,26.46,6.00),vTravel,z5,tPen\WObj:=wPaper;
    MoveL Offs(pOrigin,136.38,26.46,0.00),v60,z0,tPen\WObj:=wPaper;
    MoveL Offs(pOrigin,136.95,26.89,0.00),v40,z0,tPen\WObj:=wPaper;
    MoveL Offs(pOrigin,138.01,26.89,0.00),v40,z0,tPen\WObj:=wPaper;
    MoveL Offs(pOrigin,138.79,25.90,0.00),v40,z0,tPen\WObj:=wPaper;
    MoveL Offs(pOrigin,136.74,25.83,0.00),v40,z0,tPen\WObj:=wPaper;
    MoveL Offs(pOrigin,136.38,26.46,0.00),v40,fine,tPen\WObj:=wPaper;
    MoveL Offs(pOrigin,136.38,26.46,6.00),v60,z5,tPen\WObj:=wPaper;
    MoveL Offs(pOrigin,138.86,26.04,6.00),vTravel,z5,tPen\WObj:=wPaper;
    MoveL Offs(pOrigin,138.86,26.04,0.00),v60,z0,tPen\WObj:=wPaper;
    MoveL Offs(pOrigin,140.35,25.90,0.00),v40,z0,tPen\WObj:=wPaper;
    MoveL Offs(pOrigin,141.41,26.46,0.00),v40,z0,tPen\WObj:=wPaper;
    MoveL Offs(pOrigin,142.90,26.46,0.00),v40,z0,tPen\WObj:=wPaper;
    MoveL Offs(pOrigin,144.18,26.18,0.00),v40,z0,tPen\WObj:=wPaper;
    MoveL Offs(pOrigin,145.02,25.40,0.00),v40,z0,tPen\WObj:=wPaper;
    MoveL Offs(pOrigin,147.15,25.19,0.00),v40,z0,tPen\WObj:=wPaper;
    MoveL Offs(pOrigin,148.00,25.75,0.00),v40,z0,tPen\WObj:=wPaper;
    MoveL Offs(pOrigin,148.85,25.83,0.00),v40,z0,tPen\WObj:=wPaper;
    MoveL Offs(pOrigin,149.70,25.19,0.00),v40,z0,tPen\WObj:=wPaper;
    MoveL Offs(pOrigin,149.70,25.19,0.00),v40,z0,tPen\WObj:=wPaper;
    MoveL Offs(pOrigin,150.34,25.61,0.00),v40,z0,tPen\WObj:=wPaper;
    MoveL Offs(pOrigin,153.31,25.40,0.00),v40,z0,tPen\WObj:=wPaper;
    MoveL Offs(pOrigin,153.95,24.76,0.00),v40,z0,tPen\WObj:=wPaper;
    MoveL Offs(pOrigin,154.80,24.98,0.00),v40,z0,tPen\WObj:=wPaper;
    MoveL Offs(pOrigin,154.45,24.55,0.00),v40,z0,tPen\WObj:=wPaper;
    MoveL Offs(pOrigin,154.59,24.20,0.00),v40,z0,tPen\WObj:=wPaper;
    MoveL Offs(pOrigin,156.29,23.91,0.00),v40,fine,tPen\WObj:=wPaper;
    MoveL Offs(pOrigin,156.29,23.91,6.00),v60,z5,tPen\WObj:=wPaper;
    MoveL Offs(pOrigin,154.92,22.30,6.00),vTravel,z5,tPen\WObj:=wPaper;
    MoveL Offs(pOrigin,154.92,22.30,0.00),v60,z0,tPen\WObj:=wPaper;
    MoveL Offs(pOrigin,158.53,25.91,0.00),v40,z0,tPen\WObj:=wPaper;
    MoveL Offs(pOrigin,158.99,26.44,0.00),v40,z0,tPen\WObj:=wPaper;
    MoveL Offs(pOrigin,168.31,17.12,0.00),v40,z0,tPen\WObj:=wPaper;
    MoveL Offs(pOrigin,168.54,18.00,0.00),v40,z0,tPen\WObj:=wPaper;
    MoveL Offs(pOrigin,172.60,22.05,0.00),v40,fine,tPen\WObj:=wPaper;
    MoveL Offs(pOrigin,172.60,22.05,6.00),v60,z5,tPen\WObj:=wPaper;
    MoveL Offs(pOrigin,172.45,23.40,6.00),vTravel,z5,tPen\WObj:=wPaper;
    MoveL Offs(pOrigin,172.45,23.40,0.00),v60,z0,tPen\WObj:=wPaper;
    MoveL Offs(pOrigin,173.50,24.45,0.00),v40,z0,tPen\WObj:=wPaper;
    MoveL Offs(pOrigin,173.98,24.90,0.00),v40,z0,tPen\WObj:=wPaper;
    MoveL Offs(pOrigin,183.14,15.73,0.00),v40,z0,tPen\WObj:=wPaper;
    MoveL Offs(pOrigin,183.21,16.25,0.00),v40,z0,tPen\WObj:=wPaper;
    MoveL Offs(pOrigin,187.42,20.45,0.00),v40,fine,tPen\WObj:=wPaper;
  ENDPROC

  PROC DrawPart90()
    MoveL Offs(pOrigin,187.42,20.45,6.00),v60,z5,tPen\WObj:=wPaper;
    MoveL Offs(pOrigin,186.07,20.60,6.00),vTravel,z5,tPen\WObj:=wPaper;
    MoveL Offs(pOrigin,186.07,20.60,0.00),v60,z0,tPen\WObj:=wPaper;
    MoveL Offs(pOrigin,182.02,16.54,0.00),v40,z0,tPen\WObj:=wPaper;
    MoveL Offs(pOrigin,181.49,15.89,0.00),v40,z0,tPen\WObj:=wPaper;
    MoveL Offs(pOrigin,172.33,25.05,0.00),v40,z0,tPen\WObj:=wPaper;
    MoveL Offs(pOrigin,172.15,24.60,0.00),v40,z0,tPen\WObj:=wPaper;
    MoveL Offs(pOrigin,171.25,23.70,0.00),v40,z0,tPen\WObj:=wPaper;
    MoveL Offs(pOrigin,170.66,24.60,0.00),v40,z0,tPen\WObj:=wPaper;
    MoveL Offs(pOrigin,169.91,23.84,0.00),v40,z0,tPen\WObj:=wPaper;
    MoveL Offs(pOrigin,169.31,24.74,0.00),v40,z0,tPen\WObj:=wPaper;
    MoveL Offs(pOrigin,168.41,23.84,0.00),v40,fine,tPen\WObj:=wPaper;
    MoveL Offs(pOrigin,168.41,23.84,6.00),v60,z5,tPen\WObj:=wPaper;
    MoveL Offs(pOrigin,169.03,25.36,6.00),vTravel,z5,tPen\WObj:=wPaper;
    MoveL Offs(pOrigin,169.03,25.36,0.00),v60,z0,tPen\WObj:=wPaper;
    MoveL Offs(pOrigin,178.35,16.05,0.00),v40,z0,tPen\WObj:=wPaper;
    MoveL Offs(pOrigin,177.97,16.98,0.00),v40,z0,tPen\WObj:=wPaper;
    MoveL Offs(pOrigin,182.03,21.04,0.00),v40,fine,tPen\WObj:=wPaper;
    MoveL Offs(pOrigin,182.03,21.04,6.00),v60,z5,tPen\WObj:=wPaper;
    MoveL Offs(pOrigin,180.68,21.18,6.00),vTravel,z5,tPen\WObj:=wPaper;
    MoveL Offs(pOrigin,180.68,21.18,0.00),v60,z0,tPen\WObj:=wPaper;
    MoveL Offs(pOrigin,176.63,17.12,0.00),v40,z0,tPen\WObj:=wPaper;
    MoveL Offs(pOrigin,176.55,16.35,0.00),v40,z0,tPen\WObj:=wPaper;
    MoveL Offs(pOrigin,167.38,25.52,0.00),v40,z0,tPen\WObj:=wPaper;
    MoveL Offs(pOrigin,166.76,25.18,0.00),v40,z0,tPen\WObj:=wPaper;
    MoveL Offs(pOrigin,165.86,24.28,0.00),v40,fine,tPen\WObj:=wPaper;
    MoveL Offs(pOrigin,165.86,24.28,6.00),v60,z5,tPen\WObj:=wPaper;
    MoveL Offs(pOrigin,167.05,22.49,6.00),vTravel,z5,tPen\WObj:=wPaper;
    MoveL Offs(pOrigin,167.05,22.49,0.00),v60,z0,tPen\WObj:=wPaper;
    MoveL Offs(pOrigin,163.00,18.43,0.00),v40,z0,tPen\WObj:=wPaper;
    MoveL Offs(pOrigin,163.06,17.89,0.00),v40,z0,tPen\WObj:=wPaper;
    MoveL Offs(pOrigin,154.05,26.91,0.00),v40,z0,tPen\WObj:=wPaper;
    MoveL Offs(pOrigin,154.33,26.19,0.00),v40,z0,tPen\WObj:=wPaper;
    MoveL Offs(pOrigin,150.88,22.74,0.00),v40,fine,tPen\WObj:=wPaper;
    MoveL Offs(pOrigin,150.88,22.74,6.00),v60,z5,tPen\WObj:=wPaper;
    MoveL Offs(pOrigin,148.64,23.45,6.00),vTravel,z5,tPen\WObj:=wPaper;
    MoveL Offs(pOrigin,148.64,23.45,0.00),v60,z0,tPen\WObj:=wPaper;
    MoveL Offs(pOrigin,153.52,23.45,0.00),v40,fine,tPen\WObj:=wPaper;
    MoveL Offs(pOrigin,153.52,23.45,6.00),v60,z5,tPen\WObj:=wPaper;
    MoveL Offs(pOrigin,154.17,21.55,6.00),vTravel,z5,tPen\WObj:=wPaper;
    MoveL Offs(pOrigin,154.17,21.55,0.00),v60,z0,tPen\WObj:=wPaper;
    MoveL Offs(pOrigin,152.37,19.75,0.00),v40,fine,tPen\WObj:=wPaper;
    MoveL Offs(pOrigin,152.37,19.75,6.00),v60,z5,tPen\WObj:=wPaper;
    MoveL Offs(pOrigin,148.64,20.28,6.00),vTravel,z5,tPen\WObj:=wPaper;
    MoveL Offs(pOrigin,148.64,20.28,0.00),v60,z0,tPen\WObj:=wPaper;
    MoveL Offs(pOrigin,160.96,20.28,0.00),v40,fine,tPen\WObj:=wPaper;
    MoveL Offs(pOrigin,160.96,20.28,6.00),v60,z5,tPen\WObj:=wPaper;
    MoveL Offs(pOrigin,165.69,18.14,6.00),vTravel,z5,tPen\WObj:=wPaper;
    MoveL Offs(pOrigin,165.69,18.14,0.00),v60,z0,tPen\WObj:=wPaper;
    MoveL Offs(pOrigin,169.75,22.20,0.00),v40,fine,tPen\WObj:=wPaper;
    MoveL Offs(pOrigin,169.75,22.20,6.00),v60,z5,tPen\WObj:=wPaper;
    MoveL Offs(pOrigin,170.53,25.36,6.00),vTravel,z5,tPen\WObj:=wPaper;
    MoveL Offs(pOrigin,170.53,25.36,0.00),v60,z0,tPen\WObj:=wPaper;
    MoveL Offs(pOrigin,180.00,15.89,0.00),v40,z0,tPen\WObj:=wPaper;
    MoveL Offs(pOrigin,180.67,16.69,0.00),v40,z0,tPen\WObj:=wPaper;
    MoveL Offs(pOrigin,184.73,20.74,0.00),v40,fine,tPen\WObj:=wPaper;
    MoveL Offs(pOrigin,184.73,20.74,6.00),v60,z5,tPen\WObj:=wPaper;
    MoveL Offs(pOrigin,184.73,22.24,6.00),vTravel,z5,tPen\WObj:=wPaper;
    MoveL Offs(pOrigin,184.73,22.24,0.00),v60,z0,tPen\WObj:=wPaper;
    MoveL Offs(pOrigin,185.78,23.29,0.00),v40,z0,tPen\WObj:=wPaper;
    MoveL Offs(pOrigin,185.36,23.96,0.00),v40,z0,tPen\WObj:=wPaper;
    MoveL Offs(pOrigin,195.88,13.45,0.00),v40,fine,tPen\WObj:=wPaper;
    MoveL Offs(pOrigin,195.88,13.45,6.00),v60,z5,tPen\WObj:=wPaper;
    MoveL Offs(pOrigin,197.53,13.29,6.00),vTravel,z5,tPen\WObj:=wPaper;
    MoveL Offs(pOrigin,197.53,13.29,0.00),v60,z0,tPen\WObj:=wPaper;
    MoveL Offs(pOrigin,186.86,23.96,0.00),v40,z0,tPen\WObj:=wPaper;
    MoveL Offs(pOrigin,187.13,23.15,0.00),v40,z0,tPen\WObj:=wPaper;
    MoveL Offs(pOrigin,186.08,22.10,0.00),v40,fine,tPen\WObj:=wPaper;
    MoveL Offs(pOrigin,186.08,22.10,6.00),v60,z5,tPen\WObj:=wPaper;
    MoveL Offs(pOrigin,184.58,23.59,6.00),vTravel,z5,tPen\WObj:=wPaper;
    MoveL Offs(pOrigin,184.58,23.59,0.00),v60,z0,tPen\WObj:=wPaper;
    MoveL Offs(pOrigin,183.38,22.39,0.00),v40,fine,tPen\WObj:=wPaper;
    MoveL Offs(pOrigin,183.38,22.39,6.00),v60,z5,tPen\WObj:=wPaper;
    MoveL Offs(pOrigin,183.09,23.59,6.00),vTravel,z5,tPen\WObj:=wPaper;
    MoveL Offs(pOrigin,183.09,23.59,0.00),v60,z0,tPen\WObj:=wPaper;
    MoveL Offs(pOrigin,182.19,22.68,0.00),v40,fine,tPen\WObj:=wPaper;
    MoveL Offs(pOrigin,182.19,22.68,6.00),v60,z5,tPen\WObj:=wPaper;
    MoveL Offs(pOrigin,183.71,24.12,6.00),vTravel,z5,tPen\WObj:=wPaper;
    MoveL Offs(pOrigin,183.71,24.12,0.00),v60,z0,tPen\WObj:=wPaper;
    MoveL Offs(pOrigin,193.33,14.50,0.00),v40,fine,tPen\WObj:=wPaper;
    MoveL Offs(pOrigin,193.33,14.50,6.00),v60,z5,tPen\WObj:=wPaper;
    MoveL Offs(pOrigin,190.10,15.67,6.00),vTravel,z5,tPen\WObj:=wPaper;
    MoveL Offs(pOrigin,190.10,15.67,0.00),v60,z0,tPen\WObj:=wPaper;
    MoveL Offs(pOrigin,198.22,23.78,0.00),v40,z0,tPen\WObj:=wPaper;
    MoveL Offs(pOrigin,198.39,24.37,0.00),v40,z0,tPen\WObj:=wPaper;
    MoveL Offs(pOrigin,202.15,20.62,0.00),v40,z0,tPen\WObj:=wPaper;
    MoveL Offs(pOrigin,201.81,21.40,0.00),v40,z0,tPen\WObj:=wPaper;
    MoveL Offs(pOrigin,203.76,23.35,0.00),v40,z0,tPen\WObj:=wPaper;
    MoveL Offs(pOrigin,203.64,23.61,0.00),v40,z0,tPen\WObj:=wPaper;
    MoveL Offs(pOrigin,214.91,12.34,0.00),v40,z0,tPen\WObj:=wPaper;
    MoveL Offs(pOrigin,214.36,13.05,0.00),v40,z0,tPen\WObj:=wPaper;
    MoveL Offs(pOrigin,218.42,17.10,0.00),v40,fine,tPen\WObj:=wPaper;
    MoveL Offs(pOrigin,218.42,17.10,6.00),v60,z5,tPen\WObj:=wPaper;
    MoveL Offs(pOrigin,219.61,16.06,6.00),vTravel,z5,tPen\WObj:=wPaper;
    MoveL Offs(pOrigin,219.61,16.06,0.00),v60,z0,tPen\WObj:=wPaper;
    MoveL Offs(pOrigin,215.79,16.06,0.00),v40,fine,tPen\WObj:=wPaper;
    MoveL Offs(pOrigin,215.79,16.06,6.00),v60,z5,tPen\WObj:=wPaper;
    MoveL Offs(pOrigin,212.88,17.53,6.00),vTravel,z5,tPen\WObj:=wPaper;
    MoveL Offs(pOrigin,212.88,17.53,0.00),v60,z0,tPen\WObj:=wPaper;
    MoveL Offs(pOrigin,208.22,12.88,0.00),v40,z0,tPen\WObj:=wPaper;
    MoveL Offs(pOrigin,207.92,12.89,0.00),v40,z0,tPen\WObj:=wPaper;
    MoveL Offs(pOrigin,209.41,12.89,0.00),v40,z0,tPen\WObj:=wPaper;
    MoveL Offs(pOrigin,209.10,13.50,0.00),v40,z0,tPen\WObj:=wPaper;
    MoveL Offs(pOrigin,209.10,22.00,0.00),v40,z0,tPen\WObj:=wPaper;
    MoveL Offs(pOrigin,208.05,22.00,0.00),v40,z0,tPen\WObj:=wPaper;
    MoveL Offs(pOrigin,208.05,13.50,0.00),v40,z0,tPen\WObj:=wPaper;
    MoveL Offs(pOrigin,206.99,13.71,0.00),v40,z0,tPen\WObj:=wPaper;
    MoveL Offs(pOrigin,206.99,18.81,0.00),v40,z0,tPen\WObj:=wPaper;
    MoveL Offs(pOrigin,206.86,19.22,0.00),v40,z0,tPen\WObj:=wPaper;
    MoveL Offs(pOrigin,210.90,19.22,0.00),v40,z0,tPen\WObj:=wPaper;
    MoveL Offs(pOrigin,211.54,19.18,0.00),v40,z0,tPen\WObj:=wPaper;
    MoveL Offs(pOrigin,214.69,22.33,0.00),v40,z0,tPen\WObj:=wPaper;
    MoveL Offs(pOrigin,213.68,22.53,0.00),v40,z0,tPen\WObj:=wPaper;
    MoveL Offs(pOrigin,224.95,11.26,0.00),v40,z0,tPen\WObj:=wPaper;
    MoveL Offs(pOrigin,225.29,12.03,0.00),v40,z0,tPen\WObj:=wPaper;
    MoveL Offs(pOrigin,229.35,16.09,0.00),v40,fine,tPen\WObj:=wPaper;
    MoveL Offs(pOrigin,229.35,16.09,6.00),v60,z5,tPen\WObj:=wPaper;
    MoveL Offs(pOrigin,223.81,16.52,6.00),vTravel,z5,tPen\WObj:=wPaper;
    MoveL Offs(pOrigin,223.81,16.52,0.00),v60,z0,tPen\WObj:=wPaper;
    MoveL Offs(pOrigin,219.75,12.46,0.00),v40,z0,tPen\WObj:=wPaper;
  ENDPROC

  PROC DrawPart91()
    MoveL Offs(pOrigin,219.85,11.87,0.00),v40,z0,tPen\WObj:=wPaper;
    MoveL Offs(pOrigin,208.58,23.14,0.00),v40,z0,tPen\WObj:=wPaper;
    MoveL Offs(pOrigin,207.95,23.06,0.00),v40,z0,tPen\WObj:=wPaper;
    MoveL Offs(pOrigin,205.85,20.96,0.00),v40,fine,tPen\WObj:=wPaper;
    MoveL Offs(pOrigin,205.85,20.96,6.00),v60,z5,tPen\WObj:=wPaper;
    MoveL Offs(pOrigin,206.65,19.45,6.00),vTravel,z5,tPen\WObj:=wPaper;
    MoveL Offs(pOrigin,206.65,19.45,0.00),v60,z0,tPen\WObj:=wPaper;
    MoveL Offs(pOrigin,206.86,19.88,0.00),v40,z0,tPen\WObj:=wPaper;
    MoveL Offs(pOrigin,206.65,19.45,0.00),v40,fine,tPen\WObj:=wPaper;
    MoveL Offs(pOrigin,206.65,19.45,6.00),v60,z5,tPen\WObj:=wPaper;
    MoveL Offs(pOrigin,206.23,17.11,6.00),vTravel,z5,tPen\WObj:=wPaper;
    MoveL Offs(pOrigin,206.23,17.11,0.00),v60,z0,tPen\WObj:=wPaper;
    MoveL Offs(pOrigin,211.54,17.11,0.00),v40,z0,tPen\WObj:=wPaper;
    MoveL Offs(pOrigin,211.68,17.83,0.00),v40,z0,tPen\WObj:=wPaper;
    MoveL Offs(pOrigin,206.87,13.02,0.00),v40,z0,tPen\WObj:=wPaper;
    MoveL Offs(pOrigin,207.42,12.36,0.00),v40,z0,tPen\WObj:=wPaper;
    MoveL Offs(pOrigin,203.81,15.97,0.00),v40,fine,tPen\WObj:=wPaper;
    MoveL Offs(pOrigin,203.81,15.97,6.00),v60,z5,tPen\WObj:=wPaper;
    MoveL Offs(pOrigin,205.01,16.26,6.00),vTravel,z5,tPen\WObj:=wPaper;
    MoveL Offs(pOrigin,205.01,16.26,0.00),v60,z0,tPen\WObj:=wPaper;
    MoveL Offs(pOrigin,209.07,12.21,0.00),v40,fine,tPen\WObj:=wPaper;
    MoveL Offs(pOrigin,209.07,12.21,6.00),v60,z5,tPen\WObj:=wPaper;
    MoveL Offs(pOrigin,210.16,13.71,6.00),vTravel,z5,tPen\WObj:=wPaper;
    MoveL Offs(pOrigin,210.16,13.71,0.00),v60,z0,tPen\WObj:=wPaper;
    MoveL Offs(pOrigin,210.16,14.99,0.00),v40,z0,tPen\WObj:=wPaper;
    MoveL Offs(pOrigin,211.11,15.00,0.00),v40,z0,tPen\WObj:=wPaper;
    MoveL Offs(pOrigin,205.80,15.00,0.00),v40,z0,tPen\WObj:=wPaper;
    MoveL Offs(pOrigin,206.23,16.06,0.00),v40,z0,tPen\WObj:=wPaper;
    MoveL Offs(pOrigin,210.48,16.06,0.00),v40,fine,tPen\WObj:=wPaper;
    MoveL Offs(pOrigin,210.48,16.06,6.00),v60,z5,tPen\WObj:=wPaper;
    MoveL Offs(pOrigin,208.35,14.77,6.00),vTravel,z5,tPen\WObj:=wPaper;
    MoveL Offs(pOrigin,208.35,14.77,0.00),v60,z0,tPen\WObj:=wPaper;
    MoveL Offs(pOrigin,207.71,16.48,0.00),v40,z0,tPen\WObj:=wPaper;
    MoveL Offs(pOrigin,207.71,17.54,0.00),v40,z0,tPen\WObj:=wPaper;
    MoveL Offs(pOrigin,208.21,19.24,0.00),v40,z0,tPen\WObj:=wPaper;
    MoveL Offs(pOrigin,209.20,20.51,0.00),v40,fine,tPen\WObj:=wPaper;
    MoveL Offs(pOrigin,209.20,20.51,6.00),v60,z5,tPen\WObj:=wPaper;
    MoveL Offs(pOrigin,210.16,19.45,6.00),vTravel,z5,tPen\WObj:=wPaper;
    MoveL Offs(pOrigin,210.16,19.45,0.00),v60,z0,tPen\WObj:=wPaper;
    MoveL Offs(pOrigin,210.16,21.79,0.00),v40,z0,tPen\WObj:=wPaper;
    MoveL Offs(pOrigin,211.21,21.36,0.00),v40,z0,tPen\WObj:=wPaper;
    MoveL Offs(pOrigin,211.21,19.88,0.00),v40,fine,tPen\WObj:=wPaper;
    MoveL Offs(pOrigin,211.21,19.88,6.00),v60,z5,tPen\WObj:=wPaper;
    MoveL Offs(pOrigin,219.82,23.86,6.00),vTravel,z5,tPen\WObj:=wPaper;
    MoveL Offs(pOrigin,219.82,23.86,0.00),v60,z0,tPen\WObj:=wPaper;
    MoveL Offs(pOrigin,221.77,21.90,0.00),v40,fine,tPen\WObj:=wPaper;
    MoveL Offs(pOrigin,221.77,21.90,6.00),v60,z5,tPen\WObj:=wPaper;
    MoveL Offs(pOrigin,223.72,19.95,6.00),vTravel,z5,tPen\WObj:=wPaper;
    MoveL Offs(pOrigin,223.72,19.95,0.00),v60,z0,tPen\WObj:=wPaper;
    MoveL Offs(pOrigin,233.04,10.63,0.00),v40,z0,tPen\WObj:=wPaper;
    MoveL Offs(pOrigin,233.68,11.46,0.00),v40,z0,tPen\WObj:=wPaper;
    MoveL Offs(pOrigin,236.54,14.31,0.00),v40,z0,tPen\WObj:=wPaper;
    MoveL Offs(pOrigin,237.29,15.06,0.00),v40,z0,tPen\WObj:=wPaper;
    MoveL Offs(pOrigin,243.30,21.07,0.00),v40,z0,tPen\WObj:=wPaper;
    MoveL Offs(pOrigin,243.19,21.39,0.00),v40,z0,tPen\WObj:=wPaper;
    MoveL Offs(pOrigin,249.96,14.63,0.00),v40,fine,tPen\WObj:=wPaper;
    MoveL Offs(pOrigin,249.96,14.63,6.00),v60,z5,tPen\WObj:=wPaper;
    MoveL Offs(pOrigin,248.76,14.33,6.00),vTravel,z5,tPen\WObj:=wPaper;
    MoveL Offs(pOrigin,248.76,14.33,0.00),v60,z0,tPen\WObj:=wPaper;
    MoveL Offs(pOrigin,242.00,21.09,0.00),v40,z0,tPen\WObj:=wPaper;
    MoveL Offs(pOrigin,242.56,20.28,0.00),v40,z0,tPen\WObj:=wPaper;
    MoveL Offs(pOrigin,245.96,20.28,0.00),v40,fine,tPen\WObj:=wPaper;
    MoveL Offs(pOrigin,245.96,20.28,6.00),v60,z5,tPen\WObj:=wPaper;
    MoveL Offs(pOrigin,245.59,21.98,6.00),vTravel,z5,tPen\WObj:=wPaper;
    MoveL Offs(pOrigin,245.59,21.98,0.00),v60,z0,tPen\WObj:=wPaper;
    MoveL Offs(pOrigin,252.20,15.37,0.00),v40,z0,tPen\WObj:=wPaper;
    MoveL Offs(pOrigin,252.55,16.06,0.00),v40,z0,tPen\WObj:=wPaper;
    MoveL Offs(pOrigin,247.02,16.06,0.00),v40,fine,tPen\WObj:=wPaper;
    MoveL Offs(pOrigin,247.02,16.06,6.00),v60,z5,tPen\WObj:=wPaper;
    MoveL Offs(pOrigin,246.51,13.59,6.00),vTravel,z5,tPen\WObj:=wPaper;
    MoveL Offs(pOrigin,246.51,13.59,0.00),v60,z0,tPen\WObj:=wPaper;
    MoveL Offs(pOrigin,239.60,20.50,0.00),v40,fine,tPen\WObj:=wPaper;
    MoveL Offs(pOrigin,239.60,20.50,6.00),v60,z5,tPen\WObj:=wPaper;
    MoveL Offs(pOrigin,240.18,25.89,6.00),vTravel,z5,tPen\WObj:=wPaper;
    MoveL Offs(pOrigin,240.18,25.89,0.00),v60,z0,tPen\WObj:=wPaper;
    MoveL Offs(pOrigin,238.08,28.00,0.00),v40,fine,tPen\WObj:=wPaper;
    MoveL Offs(pOrigin,238.08,28.00,6.00),v60,z5,tPen\WObj:=wPaper;
    MoveL Offs(pOrigin,236.44,25.15,6.00),vTravel,z5,tPen\WObj:=wPaper;
    MoveL Offs(pOrigin,236.44,25.15,0.00),v60,z0,tPen\WObj:=wPaper;
    MoveL Offs(pOrigin,234.49,27.11,0.00),v40,fine,tPen\WObj:=wPaper;
    MoveL Offs(pOrigin,234.49,27.11,6.00),v60,z5,tPen\WObj:=wPaper;
    MoveL Offs(pOrigin,232.85,24.27,6.00),vTravel,z5,tPen\WObj:=wPaper;
    MoveL Offs(pOrigin,232.85,24.27,0.00),v60,z0,tPen\WObj:=wPaper;
    MoveL Offs(pOrigin,230.90,26.22,0.00),v40,fine,tPen\WObj:=wPaper;
    MoveL Offs(pOrigin,230.90,26.22,6.00),v60,z5,tPen\WObj:=wPaper;
    MoveL Offs(pOrigin,229.26,23.38,6.00),vTravel,z5,tPen\WObj:=wPaper;
    MoveL Offs(pOrigin,229.26,23.38,0.00),v60,z0,tPen\WObj:=wPaper;
    MoveL Offs(pOrigin,227.00,25.63,0.00),v40,fine,tPen\WObj:=wPaper;
    MoveL Offs(pOrigin,227.00,25.63,6.00),v60,z5,tPen\WObj:=wPaper;
    MoveL Offs(pOrigin,225.51,22.64,6.00),vTravel,z5,tPen\WObj:=wPaper;
    MoveL Offs(pOrigin,225.51,22.64,0.00),v60,z0,tPen\WObj:=wPaper;
    MoveL Offs(pOrigin,223.56,24.60,0.00),v40,fine,tPen\WObj:=wPaper;
    MoveL Offs(pOrigin,223.56,24.60,6.00),v60,z5,tPen\WObj:=wPaper;
    MoveL Offs(pOrigin,225.22,19.95,6.00),vTravel,z5,tPen\WObj:=wPaper;
    MoveL Offs(pOrigin,225.22,19.95,0.00),v60,z0,tPen\WObj:=wPaper;
    MoveL Offs(pOrigin,234.39,10.78,0.00),v40,fine,tPen\WObj:=wPaper;
    MoveL Offs(pOrigin,234.39,10.78,6.00),v60,z5,tPen\WObj:=wPaper;
    MoveL Offs(pOrigin,246.79,22.28,6.00),vTravel,z5,tPen\WObj:=wPaper;
    MoveL Offs(pOrigin,246.79,22.28,0.00),v60,z0,tPen\WObj:=wPaper;
    MoveL Offs(pOrigin,253.55,15.52,0.00),v40,z0,tPen\WObj:=wPaper;
    MoveL Offs(pOrigin,253.32,16.16,0.00),v40,z0,tPen\WObj:=wPaper;
    MoveL Offs(pOrigin,256.63,19.47,0.00),v40,fine,tPen\WObj:=wPaper;
    MoveL Offs(pOrigin,256.63,19.47,6.00),v60,z5,tPen\WObj:=wPaper;
    MoveL Offs(pOrigin,257.52,17.37,6.00),vTravel,z5,tPen\WObj:=wPaper;
    MoveL Offs(pOrigin,257.52,17.37,0.00),v60,z0,tPen\WObj:=wPaper;
    MoveL Offs(pOrigin,260.67,20.53,0.00),v40,fine,tPen\WObj:=wPaper;
    MoveL Offs(pOrigin,260.67,20.53,6.00),v60,z5,tPen\WObj:=wPaper;
    MoveL Offs(pOrigin,259.35,22.00,6.00),vTravel,z5,tPen\WObj:=wPaper;
    MoveL Offs(pOrigin,259.35,22.00,0.00),v60,z0,tPen\WObj:=wPaper;
    MoveL Offs(pOrigin,257.65,21.58,0.00),v40,fine,tPen\WObj:=wPaper;
    MoveL Offs(pOrigin,257.65,21.58,6.00),v60,z5,tPen\WObj:=wPaper;
    MoveL Offs(pOrigin,256.37,24.64,6.00),vTravel,z5,tPen\WObj:=wPaper;
    MoveL Offs(pOrigin,256.37,24.64,0.00),v60,z0,tPen\WObj:=wPaper;
    MoveL Offs(pOrigin,262.98,18.03,0.00),v40,fine,tPen\WObj:=wPaper;
    MoveL Offs(pOrigin,262.98,18.03,6.00),v60,z5,tPen\WObj:=wPaper;
    MoveL Offs(pOrigin,261.78,17.74,6.00),vTravel,z5,tPen\WObj:=wPaper;
    MoveL Offs(pOrigin,261.78,17.74,0.00),v60,z0,tPen\WObj:=wPaper;
    MoveL Offs(pOrigin,255.02,24.50,0.00),v40,fine,tPen\WObj:=wPaper;
    MoveL Offs(pOrigin,255.02,24.50,6.00),v60,z5,tPen\WObj:=wPaper;
    MoveL Offs(pOrigin,254.25,22.39,6.00),vTravel,z5,tPen\WObj:=wPaper;
  ENDPROC

  PROC DrawPart92()
    MoveL Offs(pOrigin,254.25,22.39,0.00),v60,z0,tPen\WObj:=wPaper;
    MoveL Offs(pOrigin,251.49,22.39,0.00),v40,z0,tPen\WObj:=wPaper;
    MoveL Offs(pOrigin,251.58,23.46,0.00),v40,z0,tPen\WObj:=wPaper;
    MoveL Offs(pOrigin,258.19,16.85,0.00),v40,fine,tPen\WObj:=wPaper;
    MoveL Offs(pOrigin,258.19,16.85,6.00),v60,z5,tPen\WObj:=wPaper;
    MoveL Offs(pOrigin,259.38,17.15,6.00),vTravel,z5,tPen\WObj:=wPaper;
    MoveL Offs(pOrigin,259.38,17.15,0.00),v60,z0,tPen\WObj:=wPaper;
    MoveL Offs(pOrigin,252.62,23.91,0.00),v40,fine,tPen\WObj:=wPaper;
    MoveL Offs(pOrigin,252.62,23.91,6.00),v60,z5,tPen\WObj:=wPaper;
    MoveL Offs(pOrigin,247.98,22.57,6.00),vTravel,z5,tPen\WObj:=wPaper;
    MoveL Offs(pOrigin,247.98,22.57,0.00),v60,z0,tPen\WObj:=wPaper;
    MoveL Offs(pOrigin,254.59,15.96,0.00),v40,fine,tPen\WObj:=wPaper;
    MoveL Offs(pOrigin,254.59,15.96,6.00),v60,z5,tPen\WObj:=wPaper;
    MoveL Offs(pOrigin,258.76,26.73,6.00),vTravel,z5,tPen\WObj:=wPaper;
    MoveL Offs(pOrigin,258.76,26.73,0.00),v60,z0,tPen\WObj:=wPaper;
    MoveL Offs(pOrigin,252.45,33.05,0.00),v40,fine,tPen\WObj:=wPaper;
    MoveL Offs(pOrigin,252.45,33.05,6.00),v60,z5,tPen\WObj:=wPaper;
    MoveL Offs(pOrigin,256.66,29.95,6.00),vTravel,z5,tPen\WObj:=wPaper;
    MoveL Offs(pOrigin,256.66,29.95,0.00),v60,z0,tPen\WObj:=wPaper;
    MoveL Offs(pOrigin,255.31,28.60,0.00),v40,z0,tPen\WObj:=wPaper;
    MoveL Offs(pOrigin,255.52,28.73,0.00),v40,z0,tPen\WObj:=wPaper;
    MoveL Offs(pOrigin,261.26,28.73,0.00),v40,z0,tPen\WObj:=wPaper;
    MoveL Offs(pOrigin,260.55,29.37,0.00),v40,z0,tPen\WObj:=wPaper;
    MoveL Offs(pOrigin,258.75,27.56,0.00),v40,fine,tPen\WObj:=wPaper;
    MoveL Offs(pOrigin,258.75,27.56,6.00),v60,z5,tPen\WObj:=wPaper;
    MoveL Offs(pOrigin,260.25,27.57,6.00),vTravel,z5,tPen\WObj:=wPaper;
    MoveL Offs(pOrigin,260.25,27.57,0.00),v60,z0,tPen\WObj:=wPaper;
    MoveL Offs(pOrigin,262.05,29.37,0.00),v40,z0,tPen\WObj:=wPaper;
    MoveL Offs(pOrigin,261.74,29.72,0.00),v40,z0,tPen\WObj:=wPaper;
    MoveL Offs(pOrigin,271.36,20.10,0.00),v40,z0,tPen\WObj:=wPaper;
    MoveL Offs(pOrigin,272.41,20.55,0.00),v40,z0,tPen\WObj:=wPaper;
    MoveL Offs(pOrigin,263.24,29.72,0.00),v40,z0,tPen\WObj:=wPaper;
    MoveL Offs(pOrigin,263.55,29.37,0.00),v40,z0,tPen\WObj:=wPaper;
    MoveL Offs(pOrigin,261.74,27.57,0.00),v40,fine,tPen\WObj:=wPaper;
    MoveL Offs(pOrigin,261.74,27.57,6.00),v60,z5,tPen\WObj:=wPaper;
    MoveL Offs(pOrigin,263.09,27.43,6.00),vTravel,z5,tPen\WObj:=wPaper;
    MoveL Offs(pOrigin,263.09,27.43,0.00),v60,z0,tPen\WObj:=wPaper;
    MoveL Offs(pOrigin,265.20,29.53,0.00),v40,z0,tPen\WObj:=wPaper;
    MoveL Offs(pOrigin,264.74,29.71,0.00),v40,z0,tPen\WObj:=wPaper;
    MoveL Offs(pOrigin,273.45,21.00,0.00),v40,fine,tPen\WObj:=wPaper;
    MoveL Offs(pOrigin,273.45,21.00,6.00),v60,z5,tPen\WObj:=wPaper;
    MoveL Offs(pOrigin,274.80,21.14,6.00),vTravel,z5,tPen\WObj:=wPaper;
    MoveL Offs(pOrigin,274.80,21.14,0.00),v60,z0,tPen\WObj:=wPaper;
    MoveL Offs(pOrigin,265.94,30.01,0.00),v40,z0,tPen\WObj:=wPaper;
    MoveL Offs(pOrigin,266.99,29.83,0.00),v40,z0,tPen\WObj:=wPaper;
    MoveL Offs(pOrigin,264.74,27.58,0.00),v40,fine,tPen\WObj:=wPaper;
    MoveL Offs(pOrigin,264.74,27.58,6.00),v60,z5,tPen\WObj:=wPaper;
    MoveL Offs(pOrigin,262.96,28.73,6.00),vTravel,z5,tPen\WObj:=wPaper;
    MoveL Offs(pOrigin,262.96,28.73,0.00),v60,z0,tPen\WObj:=wPaper;
    MoveL Offs(pOrigin,274.65,28.73,0.00),v40,z0,tPen\WObj:=wPaper;
    MoveL Offs(pOrigin,274.86,29.78,0.00),v40,z0,tPen\WObj:=wPaper;
    MoveL Offs(pOrigin,269.55,29.78,0.00),v40,z0,tPen\WObj:=wPaper;
    MoveL Offs(pOrigin,269.68,30.75,0.00),v40,z0,tPen\WObj:=wPaper;
    MoveL Offs(pOrigin,278.39,22.03,0.00),v40,fine,tPen\WObj:=wPaper;
    MoveL Offs(pOrigin,278.39,22.03,6.00),v60,z5,tPen\WObj:=wPaper;
    MoveL Offs(pOrigin,276.69,23.06,6.00),vTravel,z5,tPen\WObj:=wPaper;
    MoveL Offs(pOrigin,276.69,23.06,0.00),v60,z0,tPen\WObj:=wPaper;
    MoveL Offs(pOrigin,276.69,24.55,0.00),v40,fine,tPen\WObj:=wPaper;
    MoveL Offs(pOrigin,276.69,24.55,6.00),v60,z5,tPen\WObj:=wPaper;
    MoveL Offs(pOrigin,275.08,24.55,6.00),vTravel,z5,tPen\WObj:=wPaper;
    MoveL Offs(pOrigin,275.08,24.55,0.00),v60,z0,tPen\WObj:=wPaper;
    MoveL Offs(pOrigin,274.86,24.98,0.00),v40,z0,tPen\WObj:=wPaper;
    MoveL Offs(pOrigin,275.08,24.55,0.00),v40,z0,tPen\WObj:=wPaper;
    MoveL Offs(pOrigin,274.57,25.61,0.00),v40,z0,tPen\WObj:=wPaper;
    MoveL Offs(pOrigin,274.57,27.31,0.00),v40,fine,tPen\WObj:=wPaper;
    MoveL Offs(pOrigin,274.57,27.31,6.00),v60,z5,tPen\WObj:=wPaper;
    MoveL Offs(pOrigin,276.00,21.44,6.00),vTravel,z5,tPen\WObj:=wPaper;
    MoveL Offs(pOrigin,276.00,21.44,0.00),v60,z0,tPen\WObj:=wPaper;
    MoveL Offs(pOrigin,267.28,30.15,0.00),v40,fine,tPen\WObj:=wPaper;
    MoveL Offs(pOrigin,267.28,30.15,6.00),v60,z5,tPen\WObj:=wPaper;
    MoveL Offs(pOrigin,258.45,30.03,6.00),vTravel,z5,tPen\WObj:=wPaper;
    MoveL Offs(pOrigin,258.45,30.03,0.00),v60,z0,tPen\WObj:=wPaper;
    MoveL Offs(pOrigin,268.96,19.51,0.00),v40,fine,tPen\WObj:=wPaper;
    MoveL Offs(pOrigin,268.96,19.51,6.00),v60,z5,tPen\WObj:=wPaper;
    MoveL Offs(pOrigin,257.70,29.51,6.00),vTravel,z5,tPen\WObj:=wPaper;
    MoveL Offs(pOrigin,257.70,29.51,0.00),v60,z0,tPen\WObj:=wPaper;
    MoveL Offs(pOrigin,256.20,28.00,0.00),v40,fine,tPen\WObj:=wPaper;
    MoveL Offs(pOrigin,256.20,28.00,6.00),v60,z5,tPen\WObj:=wPaper;
    MoveL Offs(pOrigin,251.53,39.94,6.00),vTravel,z5,tPen\WObj:=wPaper;
    MoveL Offs(pOrigin,251.53,39.94,0.00),v60,z0,tPen\WObj:=wPaper;
    MoveL Offs(pOrigin,249.42,42.04,0.00),v40,z0,tPen\WObj:=wPaper;
    MoveL Offs(pOrigin,250.21,41.55,0.00),v40,z0,tPen\WObj:=wPaper;
    MoveL Offs(pOrigin,250.85,42.19,0.00),v40,z0,tPen\WObj:=wPaper;
    MoveL Offs(pOrigin,250.21,41.55,0.00),v40,fine,tPen\WObj:=wPaper;
    MoveL Offs(pOrigin,250.21,41.55,6.00),v60,z5,tPen\WObj:=wPaper;
    MoveL Offs(pOrigin,250.17,42.79,6.00),vTravel,z5,tPen\WObj:=wPaper;
    MoveL Offs(pOrigin,250.17,42.79,0.00),v60,z0,tPen\WObj:=wPaper;
    MoveL Offs(pOrigin,252.42,40.54,0.00),v40,fine,tPen\WObj:=wPaper;
    MoveL Offs(pOrigin,252.42,40.54,6.00),v60,z5,tPen\WObj:=wPaper;
    MoveL Offs(pOrigin,260.62,57.91,6.00),vTravel,z5,tPen\WObj:=wPaper;
    MoveL Offs(pOrigin,260.62,57.91,0.00),v60,z0,tPen\WObj:=wPaper;
    MoveL Offs(pOrigin,261.05,58.12,0.00),v40,z0,tPen\WObj:=wPaper;
    MoveL Offs(pOrigin,260.62,57.91,0.00),v40,fine,tPen\WObj:=wPaper;
    MoveL Offs(pOrigin,260.62,57.91,6.00),v60,z5,tPen\WObj:=wPaper;
    MoveL Offs(pOrigin,259.14,64.93,6.00),vTravel,z5,tPen\WObj:=wPaper;
    MoveL Offs(pOrigin,259.14,64.93,0.00),v60,z0,tPen\WObj:=wPaper;
    MoveL Offs(pOrigin,267.42,73.64,0.00),v40,z0,tPen\WObj:=wPaper;
    MoveL Offs(pOrigin,271.67,79.59,0.00),v40,z0,tPen\WObj:=wPaper;
    MoveL Offs(pOrigin,271.67,79.59,0.00),v40,z0,tPen\WObj:=wPaper;
    MoveL Offs(pOrigin,271.89,82.99,0.00),v40,z0,tPen\WObj:=wPaper;
    MoveL Offs(pOrigin,271.04,90.00,0.00),v40,z0,tPen\WObj:=wPaper;
    MoveL Offs(pOrigin,270.40,99.35,0.00),v40,z0,tPen\WObj:=wPaper;
    MoveL Offs(pOrigin,270.40,111.89,0.00),v40,z0,tPen\WObj:=wPaper;
    MoveL Offs(pOrigin,271.67,128.25,0.00),v40,z0,tPen\WObj:=wPaper;
    MoveL Offs(pOrigin,273.16,139.51,0.00),v40,z0,tPen\WObj:=wPaper;
    MoveL Offs(pOrigin,274.86,149.29,0.00),v40,z0,tPen\WObj:=wPaper;
    MoveL Offs(pOrigin,274.79,150.35,0.00),v40,z0,tPen\WObj:=wPaper;
    MoveL Offs(pOrigin,274.44,150.56,0.00),v40,z0,tPen\WObj:=wPaper;
    MoveL Offs(pOrigin,274.44,150.56,0.00),v40,z0,tPen\WObj:=wPaper;
    MoveL Offs(pOrigin,275.50,152.90,0.00),v40,z0,tPen\WObj:=wPaper;
    MoveL Offs(pOrigin,275.08,153.34,0.00),v40,z0,tPen\WObj:=wPaper;
    MoveL Offs(pOrigin,276.77,153.34,0.00),v40,z0,tPen\WObj:=wPaper;
    MoveL Offs(pOrigin,277.41,153.75,0.00),v40,z0,tPen\WObj:=wPaper;
    MoveL Offs(pOrigin,273.05,149.39,0.00),v40,z0,tPen\WObj:=wPaper;
    MoveL Offs(pOrigin,272.16,149.23,0.00),v40,z0,tPen\WObj:=wPaper;
    MoveL Offs(pOrigin,276.37,145.02,0.00),v40,z0,tPen\WObj:=wPaper;
    MoveL Offs(pOrigin,275.88,144.76,0.00),v40,z0,tPen\WObj:=wPaper;
    MoveL Offs(pOrigin,273.03,141.90,0.00),v40,z0,tPen\WObj:=wPaper;
    MoveL Offs(pOrigin,272.49,141.44,0.00),v40,z0,tPen\WObj:=wPaper;
    MoveL Offs(pOrigin,275.49,138.43,0.00),v40,z0,tPen\WObj:=wPaper;
  ENDPROC

  PROC DrawPart93()
    MoveL Offs(pOrigin,274.97,139.36,0.00),v40,z0,tPen\WObj:=wPaper;
    MoveL Offs(pOrigin,272.11,136.51,0.00),v40,z0,tPen\WObj:=wPaper;
    MoveL Offs(pOrigin,271.75,136.20,0.00),v40,z0,tPen\WObj:=wPaper;
    MoveL Offs(pOrigin,274.61,133.34,0.00),v40,z0,tPen\WObj:=wPaper;
    MoveL Offs(pOrigin,274.05,133.97,0.00),v40,z0,tPen\WObj:=wPaper;
    MoveL Offs(pOrigin,271.50,131.41,0.00),v40,z0,tPen\WObj:=wPaper;
    MoveL Offs(pOrigin,271.17,130.81,0.00),v40,z0,tPen\WObj:=wPaper;
    MoveL Offs(pOrigin,274.02,127.95,0.00),v40,z0,tPen\WObj:=wPaper;
    MoveL Offs(pOrigin,273.58,127.52,0.00),v40,z0,tPen\WObj:=wPaper;
    MoveL Offs(pOrigin,271.03,124.97,0.00),v40,z0,tPen\WObj:=wPaper;
    MoveL Offs(pOrigin,270.44,125.57,0.00),v40,z0,tPen\WObj:=wPaper;
    MoveL Offs(pOrigin,273.44,122.56,0.00),v40,z0,tPen\WObj:=wPaper;
    MoveL Offs(pOrigin,272.97,122.43,0.00),v40,z0,tPen\WObj:=wPaper;
    MoveL Offs(pOrigin,270.57,120.02,0.00),v40,z0,tPen\WObj:=wPaper;
    MoveL Offs(pOrigin,270.00,120.02,0.00),v40,z0,tPen\WObj:=wPaper;
    MoveL Offs(pOrigin,273.01,117.02,0.00),v40,z0,tPen\WObj:=wPaper;
    MoveL Offs(pOrigin,272.81,117.78,0.00),v40,z0,tPen\WObj:=wPaper;
    MoveL Offs(pOrigin,270.10,115.08,0.00),v40,z0,tPen\WObj:=wPaper;
    MoveL Offs(pOrigin,270.82,115.32,0.00),v40,z0,tPen\WObj:=wPaper;
    MoveL Offs(pOrigin,271.89,115.32,0.00),v40,z0,tPen\WObj:=wPaper;
    MoveL Offs(pOrigin,272.50,115.99,0.00),v40,z0,tPen\WObj:=wPaper;
    MoveL Offs(pOrigin,270.10,113.58,0.00),v40,z0,tPen\WObj:=wPaper;
    MoveL Offs(pOrigin,270.82,114.26,0.00),v40,z0,tPen\WObj:=wPaper;
    MoveL Offs(pOrigin,271.89,114.26,0.00),v40,fine,tPen\WObj:=wPaper;
    MoveL Offs(pOrigin,271.89,114.26,6.00),v60,z5,tPen\WObj:=wPaper;
    MoveL Offs(pOrigin,272.86,115.67,6.00),vTravel,z5,tPen\WObj:=wPaper;
    MoveL Offs(pOrigin,272.86,115.67,0.00),v60,z0,tPen\WObj:=wPaper;
    MoveL Offs(pOrigin,269.86,118.68,0.00),v40,z0,tPen\WObj:=wPaper;
    MoveL Offs(pOrigin,270.41,118.38,0.00),v40,z0,tPen\WObj:=wPaper;
    MoveL Offs(pOrigin,272.97,120.93,0.00),v40,z0,tPen\WObj:=wPaper;
    MoveL Offs(pOrigin,273.30,121.21,0.00),v40,z0,tPen\WObj:=wPaper;
    MoveL Offs(pOrigin,270.29,124.22,0.00),v40,fine,tPen\WObj:=wPaper;
    MoveL Offs(pOrigin,270.29,124.22,6.00),v60,z5,tPen\WObj:=wPaper;
    MoveL Offs(pOrigin,271.46,123.77,6.00),vTravel,z5,tPen\WObj:=wPaper;
    MoveL Offs(pOrigin,271.46,123.77,0.00),v60,z0,tPen\WObj:=wPaper;
    MoveL Offs(pOrigin,272.52,123.77,0.00),v40,z0,tPen\WObj:=wPaper;
    MoveL Offs(pOrigin,273.12,124.08,0.00),v40,z0,tPen\WObj:=wPaper;
    MoveL Offs(pOrigin,270.57,121.52,0.00),v40,z0,tPen\WObj:=wPaper;
    MoveL Offs(pOrigin,270.00,121.52,0.00),v40,z0,tPen\WObj:=wPaper;
    MoveL Offs(pOrigin,273.01,118.52,0.00),v40,z0,tPen\WObj:=wPaper;
    MoveL Offs(pOrigin,272.10,118.49,0.00),v40,z0,tPen\WObj:=wPaper;
    MoveL Offs(pOrigin,271.04,118.49,0.00),v40,z0,tPen\WObj:=wPaper;
    MoveL Offs(pOrigin,271.04,117.43,0.00),v40,z0,tPen\WObj:=wPaper;
    MoveL Offs(pOrigin,272.10,117.43,0.00),v40,fine,tPen\WObj:=wPaper;
    MoveL Offs(pOrigin,272.10,117.43,6.00),v60,z5,tPen\WObj:=wPaper;
    MoveL Offs(pOrigin,272.31,120.60,6.00),vTravel,z5,tPen\WObj:=wPaper;
    MoveL Offs(pOrigin,272.31,120.60,0.00),v60,z0,tPen\WObj:=wPaper;
    MoveL Offs(pOrigin,271.25,120.60,0.00),v40,z0,tPen\WObj:=wPaper;
    MoveL Offs(pOrigin,271.25,121.66,0.00),v40,z0,tPen\WObj:=wPaper;
    MoveL Offs(pOrigin,272.31,121.66,0.00),v40,fine,tPen\WObj:=wPaper;
    MoveL Offs(pOrigin,272.31,121.66,6.00),v60,z5,tPen\WObj:=wPaper;
    MoveL Offs(pOrigin,273.59,123.91,6.00),vTravel,z5,tPen\WObj:=wPaper;
    MoveL Offs(pOrigin,273.59,123.91,0.00),v60,z0,tPen\WObj:=wPaper;
    MoveL Offs(pOrigin,270.58,126.91,0.00),v40,z0,tPen\WObj:=wPaper;
    MoveL Offs(pOrigin,271.19,126.62,0.00),v40,z0,tPen\WObj:=wPaper;
    MoveL Offs(pOrigin,273.89,129.32,0.00),v40,z0,tPen\WObj:=wPaper;
    MoveL Offs(pOrigin,274.17,129.30,0.00),v40,z0,tPen\WObj:=wPaper;
    MoveL Offs(pOrigin,271.17,132.30,0.00),v40,z0,tPen\WObj:=wPaper;
    MoveL Offs(pOrigin,271.65,133.06,0.00),v40,z0,tPen\WObj:=wPaper;
    MoveL Offs(pOrigin,274.36,135.77,0.00),v40,z0,tPen\WObj:=wPaper;
    MoveL Offs(pOrigin,275.05,135.89,0.00),v40,z0,tPen\WObj:=wPaper;
    MoveL Offs(pOrigin,272.19,138.74,0.00),v40,z0,tPen\WObj:=wPaper;
    MoveL Offs(pOrigin,272.57,138.46,0.00),v40,z0,tPen\WObj:=wPaper;
    MoveL Offs(pOrigin,275.12,141.01,0.00),v40,z0,tPen\WObj:=wPaper;
    MoveL Offs(pOrigin,275.63,141.28,0.00),v40,z0,tPen\WObj:=wPaper;
    MoveL Offs(pOrigin,271.12,145.79,0.00),v40,z0,tPen\WObj:=wPaper;
    MoveL Offs(pOrigin,270.68,144.74,0.00),v40,z0,tPen\WObj:=wPaper;
    MoveL Offs(pOrigin,275.64,139.78,0.00),v40,fine,tPen\WObj:=wPaper;
    MoveL Offs(pOrigin,275.64,139.78,6.00),v60,z5,tPen\WObj:=wPaper;
    MoveL Offs(pOrigin,274.65,140.66,6.00),vTravel,z5,tPen\WObj:=wPaper;
    MoveL Offs(pOrigin,274.65,140.66,0.00),v60,z0,tPen\WObj:=wPaper;
    MoveL Offs(pOrigin,273.59,140.66,0.00),v40,z0,tPen\WObj:=wPaper;
    MoveL Offs(pOrigin,273.80,141.72,0.00),v40,z0,tPen\WObj:=wPaper;
    MoveL Offs(pOrigin,274.86,141.72,0.00),v40,fine,tPen\WObj:=wPaper;
    MoveL Offs(pOrigin,274.86,141.72,6.00),v60,z5,tPen\WObj:=wPaper;
    MoveL Offs(pOrigin,275.93,142.48,6.00),vTravel,z5,tPen\WObj:=wPaper;
    MoveL Offs(pOrigin,275.93,142.48,0.00),v60,z0,tPen\WObj:=wPaper;
    MoveL Offs(pOrigin,271.42,146.98,0.00),v40,z0,tPen\WObj:=wPaper;
    MoveL Offs(pOrigin,272.15,146.99,0.00),v40,z0,tPen\WObj:=wPaper;
    MoveL Offs(pOrigin,277.11,151.95,0.00),v40,z0,tPen\WObj:=wPaper;
    MoveL Offs(pOrigin,276.77,152.28,0.00),v40,z0,tPen\WObj:=wPaper;
    MoveL Offs(pOrigin,274.86,152.28,0.00),v40,z0,tPen\WObj:=wPaper;
    MoveL Offs(pOrigin,274.86,152.26,0.00),v40,z0,tPen\WObj:=wPaper;
    MoveL Offs(pOrigin,274.65,152.90,0.00),v40,z0,tPen\WObj:=wPaper;
    MoveL Offs(pOrigin,276.35,157.57,0.00),v40,z0,tPen\WObj:=wPaper;
    MoveL Offs(pOrigin,279.75,174.36,0.00),v40,z0,tPen\WObj:=wPaper;
    MoveL Offs(pOrigin,278.55,177.55,0.00),v40,z0,tPen\WObj:=wPaper;
    MoveL Offs(pOrigin,277.48,178.61,0.00),v40,z0,tPen\WObj:=wPaper;
    MoveL Offs(pOrigin,277.84,180.31,0.00),v40,z0,tPen\WObj:=wPaper;
    MoveL Offs(pOrigin,277.27,181.38,0.00),v40,z0,tPen\WObj:=wPaper;
    MoveL Offs(pOrigin,277.20,183.71,0.00),v40,z0,tPen\WObj:=wPaper;
    MoveL Offs(pOrigin,276.21,186.69,0.00),v40,z0,tPen\WObj:=wPaper;
    MoveL Offs(pOrigin,275.08,187.82,0.00),v40,z0,tPen\WObj:=wPaper;
    MoveL Offs(pOrigin,272.95,187.96,0.00),v40,z0,tPen\WObj:=wPaper;
    MoveL Offs(pOrigin,272.95,187.96,0.00),v40,z0,tPen\WObj:=wPaper;
    MoveL Offs(pOrigin,273.02,188.60,0.00),v40,z0,tPen\WObj:=wPaper;
    MoveL Offs(pOrigin,274.01,189.02,0.00),v40,z0,tPen\WObj:=wPaper;
    MoveL Offs(pOrigin,275.29,188.88,0.00),v40,z0,tPen\WObj:=wPaper;
    MoveL Offs(pOrigin,276.77,187.96,0.00),v40,z0,tPen\WObj:=wPaper;
    MoveL Offs(pOrigin,278.05,184.99,0.00),v40,z0,tPen\WObj:=wPaper;
    MoveL Offs(pOrigin,279.82,177.34,0.00),v40,z0,tPen\WObj:=wPaper;
    MoveL Offs(pOrigin,280.39,177.20,0.00),v40,z0,tPen\WObj:=wPaper;
    MoveL Offs(pOrigin,287.61,206.45,0.00),v40,z0,tPen\WObj:=wPaper;
    MoveL Offs(pOrigin,288.67,215.38,0.00),v40,z0,tPen\WObj:=wPaper;
    MoveL Offs(pOrigin,288.67,219.41,0.00),v40,z0,tPen\WObj:=wPaper;
    MoveL Offs(pOrigin,288.25,220.90,0.00),v40,fine,tPen\WObj:=wPaper;
    MoveL Offs(pOrigin,288.25,220.90,6.00),v60,z5,tPen\WObj:=wPaper;
    MoveL Offs(pOrigin,289.52,220.92,6.00),vTravel,z5,tPen\WObj:=wPaper;
    MoveL Offs(pOrigin,289.52,220.92,0.00),v60,z0,tPen\WObj:=wPaper;
    MoveL Offs(pOrigin,286.34,220.92,0.00),v40,z0,tPen\WObj:=wPaper;
    MoveL Offs(pOrigin,286.34,219.86,0.00),v40,z0,tPen\WObj:=wPaper;
    MoveL Offs(pOrigin,289.31,219.86,0.00),v40,z0,tPen\WObj:=wPaper;
    MoveL Offs(pOrigin,289.90,220.00,0.00),v40,z0,tPen\WObj:=wPaper;
    MoveL Offs(pOrigin,287.79,217.90,0.00),v40,z0,tPen\WObj:=wPaper;
    MoveL Offs(pOrigin,287.19,218.81,0.00),v40,z0,tPen\WObj:=wPaper;
    MoveL Offs(pOrigin,285.91,218.81,0.00),v40,fine,tPen\WObj:=wPaper;
    MoveL Offs(pOrigin,285.91,218.81,6.00),v60,z5,tPen\WObj:=wPaper;
    MoveL Offs(pOrigin,284.80,217.89,6.00),vTravel,z5,tPen\WObj:=wPaper;
    MoveL Offs(pOrigin,284.80,217.89,0.00),v60,z0,tPen\WObj:=wPaper;
    MoveL Offs(pOrigin,291.26,224.35,0.00),v40,z0,tPen\WObj:=wPaper;
  ENDPROC

  PROC DrawPart94()
    MoveL Offs(pOrigin,290.80,224.09,0.00),v40,z0,tPen\WObj:=wPaper;
    MoveL Offs(pOrigin,286.55,224.09,0.00),v40,z0,tPen\WObj:=wPaper;
    MoveL Offs(pOrigin,286.55,223.88,0.00),v40,z0,tPen\WObj:=wPaper;
    MoveL Offs(pOrigin,286.90,225.36,0.00),v40,z0,tPen\WObj:=wPaper;
    MoveL Offs(pOrigin,289.31,230.68,0.00),v40,z0,tPen\WObj:=wPaper;
    MoveL Offs(pOrigin,290.59,236.20,0.00),v40,z0,tPen\WObj:=wPaper;
    MoveL Offs(pOrigin,291.01,245.12,0.00),v40,z0,tPen\WObj:=wPaper;
    MoveL Offs(pOrigin,290.38,249.38,0.00),v40,z0,tPen\WObj:=wPaper;
    MoveL Offs(pOrigin,290.38,249.38,0.00),v40,z0,tPen\WObj:=wPaper;
    MoveL Offs(pOrigin,290.16,250.23,0.00),v40,z0,tPen\WObj:=wPaper;
    MoveL Offs(pOrigin,290.80,251.71,0.00),v40,z0,tPen\WObj:=wPaper;
    MoveL Offs(pOrigin,290.80,251.71,0.00),v40,z0,tPen\WObj:=wPaper;
    MoveL Offs(pOrigin,292.00,254.48,0.00),v40,z0,tPen\WObj:=wPaper;
    MoveL Offs(pOrigin,292.08,255.54,0.00),v40,z0,tPen\WObj:=wPaper;
    MoveL Offs(pOrigin,291.44,257.45,0.00),v40,z0,tPen\WObj:=wPaper;
    MoveL Offs(pOrigin,291.58,258.73,0.00),v40,z0,tPen\WObj:=wPaper;
    MoveL Offs(pOrigin,290.38,260.42,0.00),v40,z0,tPen\WObj:=wPaper;
    MoveL Offs(pOrigin,290.16,261.05,0.00),v40,z0,tPen\WObj:=wPaper;
    MoveL Offs(pOrigin,286.76,261.05,0.00),v40,z0,tPen\WObj:=wPaper;
    MoveL Offs(pOrigin,286.28,261.18,0.00),v40,z0,tPen\WObj:=wPaper;
    MoveL Offs(pOrigin,290.94,265.84,0.00),v40,z0,tPen\WObj:=wPaper;
    MoveL Offs(pOrigin,291.88,265.41,0.00),v40,z0,tPen\WObj:=wPaper;
    MoveL Offs(pOrigin,279.86,277.43,0.00),v40,z0,tPen\WObj:=wPaper;
    MoveL Offs(pOrigin,280.49,277.79,0.00),v40,z0,tPen\WObj:=wPaper;
    MoveL Offs(pOrigin,297.62,294.92,0.00),v40,z0,tPen\WObj:=wPaper;
    MoveL Offs(pOrigin,297.18,294.84,0.00),v40,z0,tPen\WObj:=wPaper;
    MoveL Offs(pOrigin,294.41,294.84,0.00),v40,z0,tPen\WObj:=wPaper;
    MoveL Offs(pOrigin,294.41,295.27,0.00),v40,z0,tPen\WObj:=wPaper;
    MoveL Offs(pOrigin,290.59,294.42,0.00),v40,z0,tPen\WObj:=wPaper;
    MoveL Offs(pOrigin,290.59,294.42,0.00),v40,z0,tPen\WObj:=wPaper;
    MoveL Offs(pOrigin,291.01,293.86,0.00),v40,z0,tPen\WObj:=wPaper;
    MoveL Offs(pOrigin,292.08,293.79,0.00),v40,z0,tPen\WObj:=wPaper;
    MoveL Offs(pOrigin,293.99,294.35,0.00),v40,z0,tPen\WObj:=wPaper;
    MoveL Offs(pOrigin,294.41,295.06,0.00),v40,z0,tPen\WObj:=wPaper;
    MoveL Offs(pOrigin,295.26,295.27,0.00),v40,fine,tPen\WObj:=wPaper;
    MoveL Offs(pOrigin,295.26,295.27,6.00),v60,z5,tPen\WObj:=wPaper;
    MoveL Offs(pOrigin,294.64,294.21,6.00),vTravel,z5,tPen\WObj:=wPaper;
    MoveL Offs(pOrigin,294.64,294.21,0.00),v60,z0,tPen\WObj:=wPaper;
    MoveL Offs(pOrigin,294.64,292.09,0.00),v40,fine,tPen\WObj:=wPaper;
    MoveL Offs(pOrigin,294.64,292.09,6.00),v60,z5,tPen\WObj:=wPaper;
    MoveL Offs(pOrigin,293.58,291.45,6.00),vTravel,z5,tPen\WObj:=wPaper;
    MoveL Offs(pOrigin,293.58,291.45,0.00),v60,z0,tPen\WObj:=wPaper;
    MoveL Offs(pOrigin,293.58,293.58,0.00),v40,fine,tPen\WObj:=wPaper;
    MoveL Offs(pOrigin,293.58,293.58,6.00),v60,z5,tPen\WObj:=wPaper;
    MoveL Offs(pOrigin,292.50,291.88,6.00),vTravel,z5,tPen\WObj:=wPaper;
    MoveL Offs(pOrigin,292.50,291.88,0.00),v60,z0,tPen\WObj:=wPaper;
    MoveL Offs(pOrigin,291.86,291.24,0.00),v40,z0,tPen\WObj:=wPaper;
    MoveL Offs(pOrigin,289.31,291.24,0.00),v40,z0,tPen\WObj:=wPaper;
    MoveL Offs(pOrigin,288.46,290.60,0.00),v40,z0,tPen\WObj:=wPaper;
    MoveL Offs(pOrigin,288.46,290.60,0.00),v40,z0,tPen\WObj:=wPaper;
    MoveL Offs(pOrigin,288.89,289.75,0.00),v40,z0,tPen\WObj:=wPaper;
    MoveL Offs(pOrigin,290.16,289.11,0.00),v40,z0,tPen\WObj:=wPaper;
    MoveL Offs(pOrigin,290.16,289.11,0.00),v40,z0,tPen\WObj:=wPaper;
    MoveL Offs(pOrigin,290.59,288.55,0.00),v40,z0,tPen\WObj:=wPaper;
    MoveL Offs(pOrigin,291.44,288.48,0.00),v40,z0,tPen\WObj:=wPaper;
    MoveL Offs(pOrigin,293.56,289.11,0.00),v40,z0,tPen\WObj:=wPaper;
    MoveL Offs(pOrigin,295.26,291.24,0.00),v40,z0,tPen\WObj:=wPaper;
    MoveL Offs(pOrigin,296.47,291.73,0.00),v40,z0,tPen\WObj:=wPaper;
    MoveL Offs(pOrigin,296.54,292.09,0.00),v40,fine,tPen\WObj:=wPaper;
    MoveL Offs(pOrigin,296.54,292.09,6.00),v60,z5,tPen\WObj:=wPaper;
    MoveL Offs(pOrigin,297.60,292.73,6.00),vTravel,z5,tPen\WObj:=wPaper;
    MoveL Offs(pOrigin,297.60,292.73,0.00),v60,z0,tPen\WObj:=wPaper;
    MoveL Offs(pOrigin,289.10,292.73,0.00),v40,fine,tPen\WObj:=wPaper;
    MoveL Offs(pOrigin,289.10,292.73,6.00),v60,z5,tPen\WObj:=wPaper;
    MoveL Offs(pOrigin,288.04,293.58,6.00),vTravel,z5,tPen\WObj:=wPaper;
    MoveL Offs(pOrigin,288.04,293.58,0.00),v60,z0,tPen\WObj:=wPaper;
    MoveL Offs(pOrigin,288.67,292.65,0.00),v40,z0,tPen\WObj:=wPaper;
    MoveL Offs(pOrigin,290.38,292.09,0.00),v40,z0,tPen\WObj:=wPaper;
    MoveL Offs(pOrigin,292.50,291.88,0.00),v40,z0,tPen\WObj:=wPaper;
    MoveL Offs(pOrigin,291.86,291.67,0.00),v40,z0,tPen\WObj:=wPaper;
    MoveL Offs(pOrigin,297.81,291.67,0.00),v40,z0,tPen\WObj:=wPaper;
    MoveL Offs(pOrigin,298.54,291.61,0.00),v40,z0,tPen\WObj:=wPaper;
    MoveL Offs(pOrigin,286.52,303.63,0.00),v40,z0,tPen\WObj:=wPaper;
    MoveL Offs(pOrigin,287.19,304.20,0.00),v40,z0,tPen\WObj:=wPaper;
    MoveL Offs(pOrigin,287.75,302.29,0.00),v40,z0,tPen\WObj:=wPaper;
    MoveL Offs(pOrigin,289.74,300.16,0.00),v40,z0,tPen\WObj:=wPaper;
    MoveL Offs(pOrigin,289.88,299.52,0.00),v40,z0,tPen\WObj:=wPaper;
    MoveL Offs(pOrigin,289.10,299.10,0.00),v40,z0,tPen\WObj:=wPaper;
    MoveL Offs(pOrigin,289.10,299.10,0.00),v40,z0,tPen\WObj:=wPaper;
    MoveL Offs(pOrigin,289.17,298.46,0.00),v40,z0,tPen\WObj:=wPaper;
    MoveL Offs(pOrigin,289.95,297.68,0.00),v40,z0,tPen\WObj:=wPaper;
    MoveL Offs(pOrigin,290.80,297.61,0.00),v40,z0,tPen\WObj:=wPaper;
    MoveL Offs(pOrigin,291.23,298.04,0.00),v40,z0,tPen\WObj:=wPaper;
    MoveL Offs(pOrigin,291.23,298.04,0.00),v40,z0,tPen\WObj:=wPaper;
    MoveL Offs(pOrigin,290.38,299.31,0.00),v40,z0,tPen\WObj:=wPaper;
    MoveL Offs(pOrigin,289.95,299.31,0.00),v40,z0,tPen\WObj:=wPaper;
    MoveL Offs(pOrigin,290.16,300.12,0.00),v40,z0,tPen\WObj:=wPaper;
    MoveL Offs(pOrigin,296.75,300.12,0.00),v40,z0,tPen\WObj:=wPaper;
    MoveL Offs(pOrigin,297.03,300.31,0.00),v40,z0,tPen\WObj:=wPaper;
    MoveL Offs(pOrigin,279.60,282.88,0.00),v40,z0,tPen\WObj:=wPaper;
    MoveL Offs(pOrigin,278.64,283.13,0.00),v40,z0,tPen\WObj:=wPaper;
    MoveL Offs(pOrigin,293.52,268.25,0.00),v40,z0,tPen\WObj:=wPaper;
    MoveL Offs(pOrigin,294.26,269.00,0.00),v40,z0,tPen\WObj:=wPaper;
    MoveL Offs(pOrigin,278.49,284.78,0.00),v40,z0,tPen\WObj:=wPaper;
    MoveL Offs(pOrigin,279.61,284.38,0.00),v40,z0,tPen\WObj:=wPaper;
    MoveL Offs(pOrigin,296.89,301.66,0.00),v40,z0,tPen\WObj:=wPaper;
    MoveL Offs(pOrigin,297.46,301.65,0.00),v40,z0,tPen\WObj:=wPaper;
    MoveL Offs(pOrigin,284.54,314.57,0.00),v40,z0,tPen\WObj:=wPaper;
    MoveL Offs(pOrigin,284.00,314.40,0.00),v40,z0,tPen\WObj:=wPaper;
    MoveL Offs(pOrigin,282.51,314.61,0.00),v40,z0,tPen\WObj:=wPaper;
    MoveL Offs(pOrigin,282.09,314.40,0.00),v40,z0,tPen\WObj:=wPaper;
    MoveL Offs(pOrigin,282.09,314.40,0.00),v40,z0,tPen\WObj:=wPaper;
    MoveL Offs(pOrigin,281.24,314.40,0.00),v40,z0,tPen\WObj:=wPaper;
    MoveL Offs(pOrigin,280.81,313.76,0.00),v40,z0,tPen\WObj:=wPaper;
    MoveL Offs(pOrigin,280.81,313.76,0.00),v40,z0,tPen\WObj:=wPaper;
    MoveL Offs(pOrigin,279.54,313.55,0.00),v40,z0,tPen\WObj:=wPaper;
    MoveL Offs(pOrigin,279.54,313.55,0.00),v40,z0,tPen\WObj:=wPaper;
    MoveL Offs(pOrigin,278.05,312.06,0.00),v40,z0,tPen\WObj:=wPaper;
    MoveL Offs(pOrigin,274.23,311.85,0.00),v40,z0,tPen\WObj:=wPaper;
    MoveL Offs(pOrigin,273.80,312.06,0.00),v40,z0,tPen\WObj:=wPaper;
    MoveL Offs(pOrigin,273.80,312.06,0.00),v40,z0,tPen\WObj:=wPaper;
    MoveL Offs(pOrigin,274.01,312.56,0.00),v40,z0,tPen\WObj:=wPaper;
    MoveL Offs(pOrigin,276.77,313.41,0.00),v40,z0,tPen\WObj:=wPaper;
    MoveL Offs(pOrigin,277.62,314.61,0.00),v40,z0,tPen\WObj:=wPaper;
    MoveL Offs(pOrigin,277.62,315.25,0.00),v40,z0,tPen\WObj:=wPaper;
    MoveL Offs(pOrigin,276.77,315.25,0.00),v40,z0,tPen\WObj:=wPaper;
    MoveL Offs(pOrigin,272.95,313.98,0.00),v40,z0,tPen\WObj:=wPaper;
    MoveL Offs(pOrigin,270.61,313.76,0.00),v40,z0,tPen\WObj:=wPaper;
    MoveL Offs(pOrigin,270.61,313.76,0.00),v40,z0,tPen\WObj:=wPaper;
    MoveL Offs(pOrigin,271.04,314.47,0.00),v40,z0,tPen\WObj:=wPaper;
  ENDPROC

  PROC DrawPart95()
    MoveL Offs(pOrigin,273.94,315.46,0.00),v40,z0,tPen\WObj:=wPaper;
    MoveL Offs(pOrigin,274.44,316.52,0.00),v40,z0,tPen\WObj:=wPaper;
    MoveL Offs(pOrigin,274.23,317.59,0.00),v40,z0,tPen\WObj:=wPaper;
    MoveL Offs(pOrigin,274.44,319.08,0.00),v40,z0,tPen\WObj:=wPaper;
    MoveL Offs(pOrigin,274.17,319.27,0.00),v40,z0,tPen\WObj:=wPaper;
    MoveL Offs(pOrigin,264.86,309.95,0.00),v40,z0,tPen\WObj:=wPaper;
    MoveL Offs(pOrigin,265.94,309.73,0.00),v40,z0,tPen\WObj:=wPaper;
    MoveL Offs(pOrigin,266.58,310.22,0.00),v40,z0,tPen\WObj:=wPaper;
    MoveL Offs(pOrigin,268.49,310.58,0.00),v40,z0,tPen\WObj:=wPaper;
    MoveL Offs(pOrigin,272.52,310.15,0.00),v40,z0,tPen\WObj:=wPaper;
    MoveL Offs(pOrigin,273.16,309.73,0.00),v40,z0,tPen\WObj:=wPaper;
    MoveL Offs(pOrigin,274.01,309.73,0.00),v40,z0,tPen\WObj:=wPaper;
    MoveL Offs(pOrigin,274.44,309.09,0.00),v40,z0,tPen\WObj:=wPaper;
    MoveL Offs(pOrigin,275.29,309.09,0.00),v40,z0,tPen\WObj:=wPaper;
    MoveL Offs(pOrigin,275.71,309.73,0.00),v40,z0,tPen\WObj:=wPaper;
    MoveL Offs(pOrigin,275.71,309.73,0.00),v40,z0,tPen\WObj:=wPaper;
    MoveL Offs(pOrigin,277.62,310.15,0.00),v40,z0,tPen\WObj:=wPaper;
    MoveL Offs(pOrigin,277.62,310.15,0.00),v40,z0,tPen\WObj:=wPaper;
    MoveL Offs(pOrigin,282.30,311.71,0.00),v40,z0,tPen\WObj:=wPaper;
    MoveL Offs(pOrigin,282.73,312.27,0.00),v40,z0,tPen\WObj:=wPaper;
    MoveL Offs(pOrigin,282.73,312.27,0.00),v40,z0,tPen\WObj:=wPaper;
    MoveL Offs(pOrigin,281.88,312.49,0.00),v40,z0,tPen\WObj:=wPaper;
    MoveL Offs(pOrigin,279.33,311.85,0.00),v40,z0,tPen\WObj:=wPaper;
    MoveL Offs(pOrigin,278.48,312.06,0.00),v40,z0,tPen\WObj:=wPaper;
    MoveL Offs(pOrigin,277.75,312.39,0.00),v40,z0,tPen\WObj:=wPaper;
    MoveL Offs(pOrigin,271.44,306.08,0.00),v40,z0,tPen\WObj:=wPaper;
    MoveL Offs(pOrigin,272.10,306.46,0.00),v40,z0,tPen\WObj:=wPaper;
    MoveL Offs(pOrigin,278.48,306.46,0.00),v40,z0,tPen\WObj:=wPaper;
    MoveL Offs(pOrigin,278.69,306.75,0.00),v40,z0,tPen\WObj:=wPaper;
    MoveL Offs(pOrigin,279.11,306.33,0.00),v40,z0,tPen\WObj:=wPaper;
    MoveL Offs(pOrigin,280.39,306.33,0.00),v40,z0,tPen\WObj:=wPaper;
    MoveL Offs(pOrigin,281.03,306.71,0.00),v40,z0,tPen\WObj:=wPaper;
    MoveL Offs(pOrigin,275.62,301.30,0.00),v40,z0,tPen\WObj:=wPaper;
    MoveL Offs(pOrigin,275.71,302.23,0.00),v40,z0,tPen\WObj:=wPaper;
    MoveL Offs(pOrigin,281.02,302.23,0.00),v40,z0,tPen\WObj:=wPaper;
    MoveL Offs(pOrigin,281.24,302.29,0.00),v40,z0,tPen\WObj:=wPaper;
    MoveL Offs(pOrigin,282.30,302.71,0.00),v40,z0,tPen\WObj:=wPaper;
    MoveL Offs(pOrigin,283.08,302.43,0.00),v40,z0,tPen\WObj:=wPaper;
    MoveL Offs(pOrigin,283.58,301.08,0.00),v40,z0,tPen\WObj:=wPaper;
    MoveL Offs(pOrigin,285.27,301.08,0.00),v40,z0,tPen\WObj:=wPaper;
    MoveL Offs(pOrigin,285.49,301.44,0.00),v40,z0,tPen\WObj:=wPaper;
    MoveL Offs(pOrigin,285.13,302.50,0.00),v40,z0,tPen\WObj:=wPaper;
    MoveL Offs(pOrigin,284.42,303.35,0.00),v40,z0,tPen\WObj:=wPaper;
    MoveL Offs(pOrigin,283.36,303.77,0.00),v40,z0,tPen\WObj:=wPaper;
    MoveL Offs(pOrigin,281.45,303.99,0.00),v40,z0,tPen\WObj:=wPaper;
    MoveL Offs(pOrigin,280.81,303.56,0.00),v40,z0,tPen\WObj:=wPaper;
    MoveL Offs(pOrigin,280.81,303.56,0.00),v40,z0,tPen\WObj:=wPaper;
    MoveL Offs(pOrigin,280.81,302.50,0.00),v40,z0,tPen\WObj:=wPaper;
    MoveL Offs(pOrigin,281.24,302.29,0.00),v40,z0,tPen\WObj:=wPaper;
    MoveL Offs(pOrigin,281.24,302.29,0.00),v40,z0,tPen\WObj:=wPaper;
    MoveL Offs(pOrigin,281.24,300.45,0.00),v40,z0,tPen\WObj:=wPaper;
    MoveL Offs(pOrigin,283.36,301.01,0.00),v40,z0,tPen\WObj:=wPaper;
    MoveL Offs(pOrigin,283.55,300.27,0.00),v40,z0,tPen\WObj:=wPaper;
    MoveL Offs(pOrigin,278.59,295.31,0.00),v40,z0,tPen\WObj:=wPaper;
    MoveL Offs(pOrigin,278.69,295.70,0.00),v40,z0,tPen\WObj:=wPaper;
    MoveL Offs(pOrigin,277.70,297.19,0.00),v40,z0,tPen\WObj:=wPaper;
    MoveL Offs(pOrigin,277.62,298.89,0.00),v40,z0,tPen\WObj:=wPaper;
    MoveL Offs(pOrigin,277.62,298.89,0.00),v40,z0,tPen\WObj:=wPaper;
    MoveL Offs(pOrigin,280.60,299.74,0.00),v40,z0,tPen\WObj:=wPaper;
    MoveL Offs(pOrigin,280.60,299.74,0.00),v40,z0,tPen\WObj:=wPaper;
    MoveL Offs(pOrigin,281.02,298.04,0.00),v40,z0,tPen\WObj:=wPaper;
    MoveL Offs(pOrigin,282.09,297.12,0.00),v40,z0,tPen\WObj:=wPaper;
    MoveL Offs(pOrigin,283.15,296.76,0.00),v40,z0,tPen\WObj:=wPaper;
    MoveL Offs(pOrigin,283.15,296.76,0.00),v40,z0,tPen\WObj:=wPaper;
    MoveL Offs(pOrigin,283.15,295.49,0.00),v40,z0,tPen\WObj:=wPaper;
    MoveL Offs(pOrigin,283.15,295.49,0.00),v40,z0,tPen\WObj:=wPaper;
    MoveL Offs(pOrigin,282.58,294.64,0.00),v40,z0,tPen\WObj:=wPaper;
    MoveL Offs(pOrigin,284.00,292.73,0.00),v40,z0,tPen\WObj:=wPaper;
    MoveL Offs(pOrigin,285.27,292.30,0.00),v40,z0,tPen\WObj:=wPaper;
    MoveL Offs(pOrigin,285.27,292.30,0.00),v40,z0,tPen\WObj:=wPaper;
    MoveL Offs(pOrigin,284.85,294.42,0.00),v40,z0,tPen\WObj:=wPaper;
    MoveL Offs(pOrigin,285.06,294.85,0.00),v40,z0,tPen\WObj:=wPaper;
    MoveL Offs(pOrigin,284.64,294.42,0.00),v40,z0,tPen\WObj:=wPaper;
    MoveL Offs(pOrigin,283.79,294.42,0.00),v40,z0,tPen\WObj:=wPaper;
    MoveL Offs(pOrigin,283.15,295.06,0.00),v40,z0,tPen\WObj:=wPaper;
    MoveL Offs(pOrigin,283.15,295.49,0.00),v40,z0,tPen\WObj:=wPaper;
    MoveL Offs(pOrigin,284.64,295.27,0.00),v40,z0,tPen\WObj:=wPaper;
    MoveL Offs(pOrigin,285.06,294.85,0.00),v40,z0,tPen\WObj:=wPaper;
    MoveL Offs(pOrigin,286.12,294.84,0.00),v40,z0,tPen\WObj:=wPaper;
    MoveL Offs(pOrigin,288.68,294.84,0.00),v40,z0,tPen\WObj:=wPaper;
    MoveL Offs(pOrigin,288.89,295.06,0.00),v40,z0,tPen\WObj:=wPaper;
    MoveL Offs(pOrigin,288.25,295.91,0.00),v40,z0,tPen\WObj:=wPaper;
    MoveL Offs(pOrigin,285.70,297.40,0.00),v40,z0,tPen\WObj:=wPaper;
    MoveL Offs(pOrigin,285.49,297.73,0.00),v40,z0,tPen\WObj:=wPaper;
    MoveL Offs(pOrigin,279.33,291.57,0.00),v40,z0,tPen\WObj:=wPaper;
    MoveL Offs(pOrigin,280.39,291.67,0.00),v40,z0,tPen\WObj:=wPaper;
    MoveL Offs(pOrigin,285.49,291.67,0.00),v40,z0,tPen\WObj:=wPaper;
    MoveL Offs(pOrigin,285.27,292.30,0.00),v40,z0,tPen\WObj:=wPaper;
    MoveL Offs(pOrigin,286.98,291.52,0.00),v40,z0,tPen\WObj:=wPaper;
    MoveL Offs(pOrigin,288.04,290.60,0.00),v40,z0,tPen\WObj:=wPaper;
    MoveL Offs(pOrigin,288.89,291.24,0.00),v40,z0,tPen\WObj:=wPaper;
    MoveL Offs(pOrigin,289.52,290.62,0.00),v40,z0,tPen\WObj:=wPaper;
    MoveL Offs(pOrigin,298.02,290.62,0.00),v40,z0,tPen\WObj:=wPaper;
    MoveL Offs(pOrigin,298.20,291.03,0.00),v40,z0,tPen\WObj:=wPaper;
    MoveL Offs(pOrigin,281.68,274.50,0.00),v40,z0,tPen\WObj:=wPaper;
    MoveL Offs(pOrigin,282.09,274.78,0.00),v40,z0,tPen\WObj:=wPaper;
    MoveL Offs(pOrigin,299.73,274.78,0.00),v40,z0,tPen\WObj:=wPaper;
    MoveL Offs(pOrigin,299.30,274.88,0.00),v40,z0,tPen\WObj:=wPaper;
    MoveL Offs(pOrigin,299.94,274.73,0.00),v40,z0,tPen\WObj:=wPaper;
    MoveL Offs(pOrigin,300.36,275.30,0.00),v40,z0,tPen\WObj:=wPaper;
    MoveL Offs(pOrigin,300.36,276.15,0.00),v40,z0,tPen\WObj:=wPaper;
    MoveL Offs(pOrigin,299.73,276.58,0.00),v40,z0,tPen\WObj:=wPaper;
    MoveL Offs(pOrigin,299.73,276.58,0.00),v40,z0,tPen\WObj:=wPaper;
    MoveL Offs(pOrigin,299.73,277.64,0.00),v40,z0,tPen\WObj:=wPaper;
    MoveL Offs(pOrigin,298.88,279.98,0.00),v40,z0,tPen\WObj:=wPaper;
    MoveL Offs(pOrigin,299.09,281.67,0.00),v40,z0,tPen\WObj:=wPaper;
    MoveL Offs(pOrigin,299.09,281.67,0.00),v40,z0,tPen\WObj:=wPaper;
    MoveL Offs(pOrigin,299.09,282.74,0.00),v40,z0,tPen\WObj:=wPaper;
    MoveL Offs(pOrigin,298.45,283.80,0.00),v40,z0,tPen\WObj:=wPaper;
    MoveL Offs(pOrigin,298.66,287.84,0.00),v40,z0,tPen\WObj:=wPaper;
    MoveL Offs(pOrigin,298.24,292.73,0.00),v40,z0,tPen\WObj:=wPaper;
    MoveL Offs(pOrigin,297.60,294.85,0.00),v40,z0,tPen\WObj:=wPaper;
    MoveL Offs(pOrigin,297.39,300.59,0.00),v40,z0,tPen\WObj:=wPaper;
    MoveL Offs(pOrigin,296.75,302.08,0.00),v40,z0,tPen\WObj:=wPaper;
    MoveL Offs(pOrigin,296.75,304.20,0.00),v40,z0,tPen\WObj:=wPaper;
    MoveL Offs(pOrigin,296.33,305.26,0.00),v40,z0,tPen\WObj:=wPaper;
    MoveL Offs(pOrigin,294.62,305.69,0.00),v40,z0,tPen\WObj:=wPaper;
    MoveL Offs(pOrigin,294.62,305.69,0.00),v40,z0,tPen\WObj:=wPaper;
    MoveL Offs(pOrigin,293.70,310.15,0.00),v40,z0,tPen\WObj:=wPaper;
    MoveL Offs(pOrigin,292.92,310.79,0.00),v40,z0,tPen\WObj:=wPaper;
  ENDPROC

